Fanuc TP program (LS listing): FM141750.ls

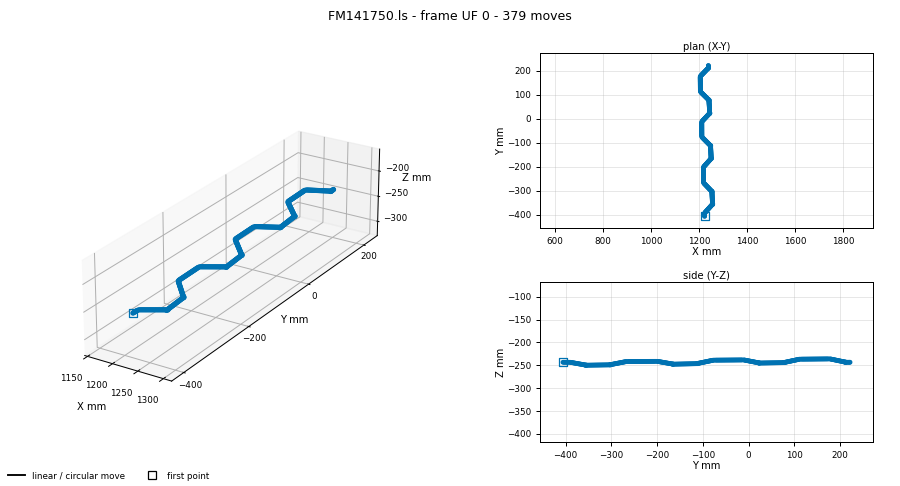
[picture p0: tool path of FM141750.ls in frame UF 0, 379 of 379 moves have a stored position in this frame; points joined in program order, loops and branches not executed]
/PROG  FM141750
/ATTR
OWNER		= MNEDITOR;
COMMENT		= "Auto FANUC move";
PROG_SIZE	= 0;
CREATE		= DATE 26-05-06  TIME 14:17:50;
MODIFIED	= DATE 26-05-06  TIME 14:17:50;
FILE_NAME	= ;
VERSION		= 0;
LINE_COUNT	= 384;
MEMORY_SIZE	= 0;
PROTECT		= READ_WRITE;
TCD:  STACK_SIZE	= 0,
      TASK_PRIORITY	= 50,
      TIME_SLICE	= 0,
      BUSY_LAMP_OFF	= 0,
      ABORT_REQUEST	= 0,
      PAUSE_REQUEST	= 0;
DEFAULT_GROUP	= 1,*,*,*,*;
CONTROL_CODE	= 00000000 00000000;
/MN
   1:  UFRAME_NUM=0 ;
   2:  UTOOL_NUM=1 ;
   3:  R[93]=10 ;
   4:  L P[1] 7mm/sec FINE ;
   5:  L P[2] 7mm/sec CNT50 ;
   6:  L P[3] 7mm/sec CNT50 ;
   7:  L P[4] 7mm/sec CNT50 ;
   8:  L P[5] 7mm/sec CNT50 ;
   9:  L P[6] 7mm/sec CNT50 ;
  10:  L P[7] 7mm/sec CNT50 ;
  11:  L P[8] 7mm/sec CNT50 ;
  12:  L P[9] 7mm/sec CNT50 ;
  13:  L P[10] 7mm/sec CNT50 ;
  14:  L P[11] 7mm/sec CNT50 ;
  15:  L P[12] 7mm/sec CNT50 ;
  16:  L P[13] 7mm/sec CNT50 ;
  17:  L P[14] 7mm/sec CNT50 ;
  18:  L P[15] 7mm/sec CNT50 ;
  19:  L P[16] 7mm/sec CNT50 ;
  20:  L P[17] 7mm/sec CNT50 ;
  21:  L P[18] 7mm/sec CNT50 ;
  22:  L P[19] 7mm/sec CNT50 ;
  23:  L P[20] 7mm/sec CNT50 ;
  24:  L P[21] 7mm/sec CNT50 ;
  25:  L P[22] 7mm/sec CNT50 ;
  26:  L P[23] 7mm/sec CNT50 ;
  27:  L P[24] 7mm/sec CNT50 ;
  28:  L P[25] 7mm/sec CNT50 ;
  29:  L P[26] 7mm/sec CNT50 ;
  30:  L P[27] 7mm/sec CNT50 ;
  31:  L P[28] 7mm/sec CNT50 ;
  32:  L P[29] 7mm/sec CNT50 ;
  33:  L P[30] 7mm/sec CNT50 ;
  34:  L P[31] 7mm/sec CNT50 ;
  35:  L P[32] 7mm/sec CNT50 ;
  36:  L P[33] 7mm/sec CNT50 ;
  37:  L P[34] 7mm/sec CNT50 ;
  38:  L P[35] 7mm/sec CNT50 ;
  39:  L P[36] 7mm/sec CNT50 ;
  40:  L P[37] 7mm/sec CNT50 ;
  41:  L P[38] 7mm/sec CNT50 ;
  42:  L P[39] 7mm/sec CNT50 ;
  43:  L P[40] 7mm/sec CNT50 ;
  44:  L P[41] 7mm/sec CNT50 ;
  45:  L P[42] 7mm/sec CNT50 ;
  46:  L P[43] 7mm/sec CNT50 ;
  47:  L P[44] 7mm/sec CNT50 ;
  48:  L P[45] 7mm/sec CNT50 ;
  49:  L P[46] 7mm/sec CNT50 ;
  50:  L P[47] 7mm/sec CNT50 ;
  51:  L P[48] 7mm/sec CNT50 ;
  52:  L P[49] 7mm/sec CNT50 ;
  53:  L P[50] 7mm/sec CNT50 ;
  54:  L P[51] 7mm/sec CNT50 ;
  55:  L P[52] 7mm/sec CNT50 ;
  56:  L P[53] 7mm/sec CNT50 ;
  57:  L P[54] 7mm/sec CNT50 ;
  58:  L P[55] 7mm/sec CNT50 ;
  59:  L P[56] 7mm/sec CNT50 ;
  60:  L P[57] 7mm/sec CNT50 ;
  61:  L P[58] 7mm/sec CNT50 ;
  62:  L P[59] 7mm/sec CNT50 ;
  63:  L P[60] 7mm/sec CNT50 ;
  64:  L P[61] 7mm/sec CNT50 ;
  65:  L P[62] 7mm/sec CNT50 ;
  66:  L P[63] 7mm/sec CNT50 ;
  67:  L P[64] 7mm/sec CNT50 ;
  68:  L P[65] 7mm/sec CNT50 ;
  69:  L P[66] 7mm/sec CNT50 ;
  70:  L P[67] 7mm/sec CNT50 ;
  71:  L P[68] 7mm/sec CNT50 ;
  72:  L P[69] 7mm/sec CNT50 ;
  73:  L P[70] 7mm/sec CNT50 ;
  74:  L P[71] 7mm/sec CNT50 ;
  75:  L P[72] 7mm/sec CNT50 ;
  76:  L P[73] 7mm/sec CNT50 ;
  77:  L P[74] 7mm/sec CNT50 ;
  78:  L P[75] 7mm/sec CNT50 ;
  79:  L P[76] 7mm/sec CNT50 ;
  80:  L P[77] 7mm/sec CNT50 ;
  81:  L P[78] 7mm/sec CNT50 ;
  82:  L P[79] 7mm/sec CNT50 ;
  83:  L P[80] 7mm/sec CNT50 ;
  84:  L P[81] 7mm/sec CNT50 ;
  85:  L P[82] 7mm/sec CNT50 ;
  86:  L P[83] 7mm/sec CNT50 ;
  87:  L P[84] 7mm/sec CNT50 ;
  88:  L P[85] 7mm/sec CNT50 ;
  89:  L P[86] 7mm/sec CNT50 ;
  90:  L P[87] 7mm/sec CNT50 ;
  91:  L P[88] 7mm/sec CNT50 ;
  92:  L P[89] 7mm/sec CNT50 ;
  93:  L P[90] 7mm/sec CNT50 ;
  94:  L P[91] 7mm/sec CNT50 ;
  95:  L P[92] 7mm/sec CNT50 ;
  96:  L P[93] 7mm/sec CNT50 ;
  97:  L P[94] 7mm/sec CNT50 ;
  98:  L P[95] 7mm/sec CNT50 ;
  99:  L P[96] 7mm/sec CNT50 ;
 100:  L P[97] 7mm/sec CNT50 ;
 101:  L P[98] 7mm/sec CNT50 ;
 102:  L P[99] 7mm/sec CNT50 ;
 103:  L P[100] 7mm/sec CNT50 ;
 104:  L P[101] 7mm/sec CNT50 ;
 105:  L P[102] 7mm/sec CNT50 ;
 106:  L P[103] 7mm/sec CNT50 ;
 107:  L P[104] 7mm/sec CNT50 ;
 108:  L P[105] 7mm/sec CNT50 ;
 109:  L P[106] 7mm/sec CNT50 ;
 110:  L P[107] 7mm/sec CNT50 ;
 111:  L P[108] 7mm/sec CNT50 ;
 112:  L P[109] 7mm/sec CNT50 ;
 113:  L P[110] 7mm/sec CNT50 ;
 114:  L P[111] 7mm/sec CNT50 ;
 115:  L P[112] 7mm/sec CNT50 ;
 116:  L P[113] 7mm/sec CNT50 ;
 117:  L P[114] 7mm/sec CNT50 ;
 118:  L P[115] 7mm/sec CNT50 ;
 119:  L P[116] 7mm/sec CNT50 ;
 120:  L P[117] 7mm/sec CNT50 ;
 121:  L P[118] 7mm/sec CNT50 ;
 122:  L P[119] 7mm/sec CNT50 ;
 123:  L P[120] 7mm/sec CNT50 ;
 124:  L P[121] 7mm/sec CNT50 ;
 125:  L P[122] 7mm/sec CNT50 ;
 126:  L P[123] 7mm/sec CNT50 ;
 127:  L P[124] 7mm/sec CNT50 ;
 128:  L P[125] 7mm/sec CNT50 ;
 129:  L P[126] 7mm/sec CNT50 ;
 130:  L P[127] 7mm/sec CNT50 ;
 131:  L P[128] 7mm/sec CNT50 ;
 132:  L P[129] 7mm/sec CNT50 ;
 133:  L P[130] 7mm/sec CNT50 ;
 134:  L P[131] 7mm/sec CNT50 ;
 135:  L P[132] 7mm/sec CNT50 ;
 136:  L P[133] 7mm/sec CNT50 ;
 137:  L P[134] 7mm/sec CNT50 ;
 138:  L P[135] 7mm/sec CNT50 ;
 139:  L P[136] 7mm/sec CNT50 ;
 140:  L P[137] 7mm/sec CNT50 ;
 141:  L P[138] 7mm/sec CNT50 ;
 142:  L P[139] 7mm/sec CNT50 ;
 143:  L P[140] 7mm/sec CNT50 ;
 144:  L P[141] 7mm/sec CNT50 ;
 145:  L P[142] 7mm/sec CNT50 ;
 146:  L P[143] 7mm/sec CNT50 ;
 147:  L P[144] 7mm/sec CNT50 ;
 148:  L P[145] 7mm/sec CNT50 ;
 149:  L P[146] 7mm/sec CNT50 ;
 150:  L P[147] 7mm/sec CNT50 ;
 151:  L P[148] 7mm/sec CNT50 ;
 152:  L P[149] 7mm/sec CNT50 ;
 153:  L P[150] 7mm/sec CNT50 ;
 154:  L P[151] 7mm/sec CNT50 ;
 155:  L P[152] 7mm/sec CNT50 ;
 156:  L P[153] 7mm/sec CNT50 ;
 157:  L P[154] 7mm/sec CNT50 ;
 158:  L P[155] 7mm/sec CNT50 ;
 159:  L P[156] 7mm/sec CNT50 ;
 160:  L P[157] 7mm/sec CNT50 ;
 161:  L P[158] 7mm/sec CNT50 ;
 162:  L P[159] 7mm/sec CNT50 ;
 163:  L P[160] 7mm/sec CNT50 ;
 164:  L P[161] 7mm/sec CNT50 ;
 165:  L P[162] 7mm/sec CNT50 ;
 166:  L P[163] 7mm/sec CNT50 ;
 167:  L P[164] 7mm/sec CNT50 ;
 168:  L P[165] 7mm/sec CNT50 ;
 169:  L P[166] 7mm/sec CNT50 ;
 170:  L P[167] 7mm/sec CNT50 ;
 171:  L P[168] 7mm/sec CNT50 ;
 172:  L P[169] 7mm/sec CNT50 ;
 173:  L P[170] 7mm/sec CNT50 ;
 174:  L P[171] 7mm/sec CNT50 ;
 175:  L P[172] 7mm/sec CNT50 ;
 176:  L P[173] 7mm/sec CNT50 ;
 177:  L P[174] 7mm/sec CNT50 ;
 178:  L P[175] 7mm/sec CNT50 ;
 179:  L P[176] 7mm/sec CNT50 ;
 180:  L P[177] 7mm/sec CNT50 ;
 181:  L P[178] 7mm/sec CNT50 ;
 182:  L P[179] 7mm/sec CNT50 ;
 183:  L P[180] 7mm/sec CNT50 ;
 184:  L P[181] 7mm/sec CNT50 ;
 185:  L P[182] 7mm/sec CNT50 ;
 186:  L P[183] 7mm/sec CNT50 ;
 187:  L P[184] 7mm/sec CNT50 ;
 188:  L P[185] 7mm/sec CNT50 ;
 189:  L P[186] 7mm/sec CNT50 ;
 190:  L P[187] 7mm/sec CNT50 ;
 191:  L P[188] 7mm/sec CNT50 ;
 192:  L P[189] 7mm/sec CNT50 ;
 193:  L P[190] 7mm/sec CNT50 ;
 194:  L P[191] 7mm/sec CNT50 ;
 195:  L P[192] 7mm/sec CNT50 ;
 196:  L P[193] 7mm/sec CNT50 ;
 197:  L P[194] 7mm/sec CNT50 ;
 198:  L P[195] 7mm/sec CNT50 ;
 199:  L P[196] 7mm/sec CNT50 ;
 200:  L P[197] 7mm/sec CNT50 ;
 201:  L P[198] 7mm/sec CNT50 ;
 202:  L P[199] 7mm/sec CNT50 ;
 203:  L P[200] 7mm/sec CNT50 ;
 204:  L P[201] 7mm/sec CNT50 ;
 205:  L P[202] 7mm/sec CNT50 ;
 206:  L P[203] 7mm/sec CNT50 ;
 207:  L P[204] 7mm/sec CNT50 ;
 208:  L P[205] 7mm/sec CNT50 ;
 209:  L P[206] 7mm/sec CNT50 ;
 210:  L P[207] 7mm/sec CNT50 ;
 211:  L P[208] 7mm/sec CNT50 ;
 212:  L P[209] 7mm/sec CNT50 ;
 213:  L P[210] 7mm/sec CNT50 ;
 214:  L P[211] 7mm/sec CNT50 ;
 215:  L P[212] 7mm/sec CNT50 ;
 216:  L P[213] 7mm/sec CNT50 ;
 217:  L P[214] 7mm/sec CNT50 ;
 218:  L P[215] 7mm/sec CNT50 ;
 219:  L P[216] 7mm/sec CNT50 ;
 220:  L P[217] 7mm/sec CNT50 ;
 221:  L P[218] 7mm/sec CNT50 ;
 222:  L P[219] 7mm/sec CNT50 ;
 223:  L P[220] 7mm/sec CNT50 ;
 224:  L P[221] 7mm/sec CNT50 ;
 225:  L P[222] 7mm/sec CNT50 ;
 226:  L P[223] 7mm/sec CNT50 ;
 227:  L P[224] 7mm/sec CNT50 ;
 228:  L P[225] 7mm/sec CNT50 ;
 229:  L P[226] 7mm/sec CNT50 ;
 230:  L P[227] 7mm/sec CNT50 ;
 231:  L P[228] 7mm/sec CNT50 ;
 232:  L P[229] 7mm/sec CNT50 ;
 233:  L P[230] 7mm/sec CNT50 ;
 234:  L P[231] 7mm/sec CNT50 ;
 235:  L P[232] 7mm/sec CNT50 ;
 236:  L P[233] 7mm/sec CNT50 ;
 237:  L P[234] 7mm/sec CNT50 ;
 238:  L P[235] 7mm/sec CNT50 ;
 239:  L P[236] 7mm/sec CNT50 ;
 240:  L P[237] 7mm/sec CNT50 ;
 241:  L P[238] 7mm/sec CNT50 ;
 242:  L P[239] 7mm/sec CNT50 ;
 243:  L P[240] 7mm/sec CNT50 ;
 244:  L P[241] 7mm/sec CNT50 ;
 245:  L P[242] 7mm/sec CNT50 ;
 246:  L P[243] 7mm/sec CNT50 ;
 247:  L P[244] 7mm/sec CNT50 ;
 248:  L P[245] 7mm/sec CNT50 ;
 249:  L P[246] 7mm/sec CNT50 ;
 250:  L P[247] 7mm/sec CNT50 ;
 251:  L P[248] 7mm/sec CNT50 ;
 252:  L P[249] 7mm/sec CNT50 ;
 253:  L P[250] 7mm/sec CNT50 ;
 254:  L P[251] 7mm/sec CNT50 ;
 255:  L P[252] 7mm/sec CNT50 ;
 256:  L P[253] 7mm/sec CNT50 ;
 257:  L P[254] 7mm/sec CNT50 ;
 258:  L P[255] 7mm/sec CNT50 ;
 259:  L P[256] 7mm/sec CNT50 ;
 260:  L P[257] 7mm/sec CNT50 ;
 261:  L P[258] 7mm/sec CNT50 ;
 262:  L P[259] 7mm/sec CNT50 ;
 263:  L P[260] 7mm/sec CNT50 ;
 264:  L P[261] 7mm/sec CNT50 ;
 265:  L P[262] 7mm/sec CNT50 ;
 266:  L P[263] 7mm/sec CNT50 ;
 267:  L P[264] 7mm/sec CNT50 ;
 268:  L P[265] 7mm/sec CNT50 ;
 269:  L P[266] 7mm/sec CNT50 ;
 270:  L P[267] 7mm/sec CNT50 ;
 271:  L P[268] 7mm/sec CNT50 ;
 272:  L P[269] 7mm/sec CNT50 ;
 273:  L P[270] 7mm/sec CNT50 ;
 274:  L P[271] 7mm/sec CNT50 ;
 275:  L P[272] 7mm/sec CNT50 ;
 276:  L P[273] 7mm/sec CNT50 ;
 277:  L P[274] 7mm/sec CNT50 ;
 278:  L P[275] 7mm/sec CNT50 ;
 279:  L P[276] 7mm/sec CNT50 ;
 280:  L P[277] 7mm/sec CNT50 ;
 281:  L P[278] 7mm/sec CNT50 ;
 282:  L P[279] 7mm/sec CNT50 ;
 283:  L P[280] 7mm/sec CNT50 ;
 284:  L P[281] 7mm/sec CNT50 ;
 285:  L P[282] 7mm/sec CNT50 ;
 286:  L P[283] 7mm/sec CNT50 ;
 287:  L P[284] 7mm/sec CNT50 ;
 288:  L P[285] 7mm/sec CNT50 ;
 289:  L P[286] 7mm/sec CNT50 ;
 290:  L P[287] 7mm/sec CNT50 ;
 291:  L P[288] 7mm/sec CNT50 ;
 292:  L P[289] 7mm/sec CNT50 ;
 293:  L P[290] 7mm/sec CNT50 ;
 294:  L P[291] 7mm/sec CNT50 ;
 295:  L P[292] 7mm/sec CNT50 ;
 296:  L P[293] 7mm/sec CNT50 ;
 297:  L P[294] 7mm/sec CNT50 ;
 298:  L P[295] 7mm/sec CNT50 ;
 299:  L P[296] 7mm/sec CNT50 ;
 300:  L P[297] 7mm/sec CNT50 ;
 301:  L P[298] 7mm/sec CNT50 ;
 302:  L P[299] 7mm/sec CNT50 ;
 303:  L P[300] 7mm/sec CNT50 ;
 304:  L P[301] 7mm/sec CNT50 ;
 305:  L P[302] 7mm/sec CNT50 ;
 306:  L P[303] 7mm/sec CNT50 ;
 307:  L P[304] 7mm/sec CNT50 ;
 308:  L P[305] 7mm/sec CNT50 ;
 309:  L P[306] 7mm/sec CNT50 ;
 310:  L P[307] 7mm/sec CNT50 ;
 311:  L P[308] 7mm/sec CNT50 ;
 312:  L P[309] 7mm/sec CNT50 ;
 313:  L P[310] 7mm/sec CNT50 ;
 314:  L P[311] 7mm/sec CNT50 ;
 315:  L P[312] 7mm/sec CNT50 ;
 316:  L P[313] 7mm/sec CNT50 ;
 317:  L P[314] 7mm/sec CNT50 ;
 318:  L P[315] 7mm/sec CNT50 ;
 319:  L P[316] 7mm/sec CNT50 ;
 320:  L P[317] 7mm/sec CNT50 ;
 321:  L P[318] 7mm/sec CNT50 ;
 322:  L P[319] 7mm/sec CNT50 ;
 323:  L P[320] 7mm/sec CNT50 ;
 324:  L P[321] 7mm/sec CNT50 ;
 325:  L P[322] 7mm/sec CNT50 ;
 326:  L P[323] 7mm/sec CNT50 ;
 327:  L P[324] 7mm/sec CNT50 ;
 328:  L P[325] 7mm/sec CNT50 ;
 329:  L P[326] 7mm/sec CNT50 ;
 330:  L P[327] 7mm/sec CNT50 ;
 331:  L P[328] 7mm/sec CNT50 ;
 332:  L P[329] 7mm/sec CNT50 ;
 333:  L P[330] 7mm/sec CNT50 ;
 334:  L P[331] 7mm/sec CNT50 ;
 335:  L P[332] 7mm/sec CNT50 ;
 336:  L P[333] 7mm/sec CNT50 ;
 337:  L P[334] 7mm/sec CNT50 ;
 338:  L P[335] 7mm/sec CNT50 ;
 339:  L P[336] 7mm/sec CNT50 ;
 340:  L P[337] 7mm/sec CNT50 ;
 341:  L P[338] 7mm/sec CNT50 ;
 342:  L P[339] 7mm/sec CNT50 ;
 343:  L P[340] 7mm/sec CNT50 ;
 344:  L P[341] 7mm/sec CNT50 ;
 345:  L P[342] 7mm/sec CNT50 ;
 346:  L P[343] 7mm/sec CNT50 ;
 347:  L P[344] 7mm/sec CNT50 ;
 348:  L P[345] 7mm/sec CNT50 ;
 349:  L P[346] 7mm/sec CNT50 ;
 350:  L P[347] 7mm/sec CNT50 ;
 351:  L P[348] 7mm/sec CNT50 ;
 352:  L P[349] 7mm/sec CNT50 ;
 353:  L P[350] 7mm/sec CNT50 ;
 354:  L P[351] 7mm/sec CNT50 ;
 355:  L P[352] 7mm/sec CNT50 ;
 356:  L P[353] 7mm/sec CNT50 ;
 357:  L P[354] 7mm/sec CNT50 ;
 358:  L P[355] 7mm/sec CNT50 ;
 359:  L P[356] 7mm/sec CNT50 ;
 360:  L P[357] 7mm/sec CNT50 ;
 361:  L P[358] 7mm/sec CNT50 ;
 362:  L P[359] 7mm/sec CNT50 ;
 363:  L P[360] 7mm/sec CNT50 ;
 364:  L P[361] 7mm/sec CNT50 ;
 365:  L P[362] 7mm/sec CNT50 ;
 366:  L P[363] 7mm/sec CNT50 ;
 367:  L P[364] 7mm/sec CNT50 ;
 368:  L P[365] 7mm/sec CNT50 ;
 369:  L P[366] 7mm/sec CNT50 ;
 370:  L P[367] 7mm/sec CNT50 ;
 371:  L P[368] 7mm/sec CNT50 ;
 372:  L P[369] 7mm/sec CNT50 ;
 373:  L P[370] 7mm/sec CNT50 ;
 374:  L P[371] 7mm/sec CNT50 ;
 375:  L P[372] 7mm/sec CNT50 ;
 376:  L P[373] 7mm/sec CNT50 ;
 377:  L P[374] 7mm/sec CNT50 ;
 378:  L P[375] 7mm/sec CNT50 ;
 379:  L P[376] 7mm/sec CNT50 ;
 380:  L P[377] 7mm/sec CNT50 ;
 381:  L P[378] 7mm/sec CNT50 ;
 382:  L P[379] 7mm/sec FINE ;
 383:  R[93]=1 ;
 384:  END ;
/POS
P[1]{
   GP1:
	UF : 0, UT : 1,		CONFIG : 'N U T, 0, 0, 0',
	X = 1222.210  mm,	Y = -405.958  mm,	Z = -243.379  mm,
	W = 0.000 deg,	P = 30.000 deg,	R = 178.529 deg
};
P[2]{
   GP1:
	UF : 0, UT : 1,		CONFIG : 'N U T, 0, 0, 0',
	X = 1222.261  mm,	Y = -403.959  mm,	Z = -243.380  mm,
	W = 0.000 deg,	P = 30.000 deg,	R = 178.529 deg
};
P[3]{
   GP1:
	UF : 0, UT : 1,		CONFIG : 'N U T, 0, 0, 0',
	X = 1222.312  mm,	Y = -401.960  mm,	Z = -243.381  mm,
	W = 0.000 deg,	P = 30.000 deg,	R = 170.399 deg
};
P[4]{
   GP1:
	UF : 0, UT : 1,		CONFIG : 'N U T, 0, 0, 0',
	X = 1222.364  mm,	Y = -399.960  mm,	Z = -243.383  mm,
	W = 0.000 deg,	P = 30.000 deg,	R = 162.269 deg
};
P[5]{
   GP1:
	UF : 0, UT : 1,		CONFIG : 'N U T, 0, 0, 0',
	X = 1222.415  mm,	Y = -397.961  mm,	Z = -243.384  mm,
	W = 0.000 deg,	P = 30.000 deg,	R = 154.139 deg
};
P[6]{
   GP1:
	UF : 0, UT : 1,		CONFIG : 'N U T, 0, 0, 0',
	X = 1222.466  mm,	Y = -395.962  mm,	Z = -243.385  mm,
	W = 0.000 deg,	P = 30.000 deg,	R = 146.009 deg
};
P[7]{
   GP1:
	UF : 0, UT : 1,		CONFIG : 'N U T, 0, 0, 0',
	X = 1222.518  mm,	Y = -393.962  mm,	Z = -243.387  mm,
	W = 0.000 deg,	P = 30.000 deg,	R = 137.880 deg
};
P[8]{
   GP1:
	UF : 0, UT : 1,		CONFIG : 'N U T, 0, 0, 0',
	X = 1223.380  mm,	Y = -390.882  mm,	Z = -243.387  mm,
	W = 0.000 deg,	P = 30.000 deg,	R = 137.880 deg
};
P[9]{
   GP1:
	UF : 0, UT : 1,		CONFIG : 'N U T, 0, 0, 0',
	X = 1224.872  mm,	Y = -389.157  mm,	Z = -243.595  mm,
	W = 0.000 deg,	P = 30.000 deg,	R = 137.880 deg
};
P[10]{
   GP1:
	UF : 0, UT : 1,		CONFIG : 'N U T, 0, 0, 0',
	X = 1226.202  mm,	Y = -387.686  mm,	Z = -243.857  mm,
	W = 0.000 deg,	P = 30.000 deg,	R = 137.880 deg
};
P[11]{
   GP1:
	UF : 0, UT : 1,		CONFIG : 'N U T, 0, 0, 0',
	X = 1227.531  mm,	Y = -386.216  mm,	Z = -244.119  mm,
	W = 0.000 deg,	P = 30.000 deg,	R = 137.880 deg
};
P[12]{
   GP1:
	UF : 0, UT : 1,		CONFIG : 'N U T, 0, 0, 0',
	X = 1228.861  mm,	Y = -384.745  mm,	Z = -244.381  mm,
	W = 0.000 deg,	P = 30.000 deg,	R = 137.880 deg
};
P[13]{
   GP1:
	UF : 0, UT : 1,		CONFIG : 'N U T, 0, 0, 0',
	X = 1230.191  mm,	Y = -383.274  mm,	Z = -244.643  mm,
	W = 0.000 deg,	P = 30.000 deg,	R = 137.880 deg
};
P[14]{
   GP1:
	UF : 0, UT : 1,		CONFIG : 'N U T, 0, 0, 0',
	X = 1231.521  mm,	Y = -381.804  mm,	Z = -244.905  mm,
	W = 0.000 deg,	P = 30.000 deg,	R = 137.880 deg
};
P[15]{
   GP1:
	UF : 0, UT : 1,		CONFIG : 'N U T, 0, 0, 0',
	X = 1232.851  mm,	Y = -380.333  mm,	Z = -245.167  mm,
	W = 0.000 deg,	P = 30.000 deg,	R = 137.880 deg
};
P[16]{
   GP1:
	UF : 0, UT : 1,		CONFIG : 'N U T, 0, 0, 0',
	X = 1234.181  mm,	Y = -378.862  mm,	Z = -245.429  mm,
	W = 0.000 deg,	P = 30.000 deg,	R = 137.880 deg
};
P[17]{
   GP1:
	UF : 0, UT : 1,		CONFIG : 'N U T, 0, 0, 0',
	X = 1235.510  mm,	Y = -377.392  mm,	Z = -245.692  mm,
	W = 0.000 deg,	P = 30.000 deg,	R = 137.880 deg
};
P[18]{
   GP1:
	UF : 0, UT : 1,		CONFIG : 'N U T, 0, 0, 0',
	X = 1236.840  mm,	Y = -375.921  mm,	Z = -245.954  mm,
	W = 0.000 deg,	P = 30.000 deg,	R = 137.880 deg
};
P[19]{
   GP1:
	UF : 0, UT : 1,		CONFIG : 'N U T, 0, 0, 0',
	X = 1238.170  mm,	Y = -374.450  mm,	Z = -246.216  mm,
	W = 0.000 deg,	P = 30.000 deg,	R = 137.880 deg
};
P[20]{
   GP1:
	UF : 0, UT : 1,		CONFIG : 'N U T, 0, 0, 0',
	X = 1239.500  mm,	Y = -372.979  mm,	Z = -246.478  mm,
	W = 0.000 deg,	P = 30.000 deg,	R = 137.880 deg
};
P[21]{
   GP1:
	UF : 0, UT : 1,		CONFIG : 'N U T, 0, 0, 0',
	X = 1240.830  mm,	Y = -371.509  mm,	Z = -246.740  mm,
	W = 0.000 deg,	P = 30.000 deg,	R = 137.880 deg
};
P[22]{
   GP1:
	UF : 0, UT : 1,		CONFIG : 'N U T, 0, 0, 0',
	X = 1242.159  mm,	Y = -370.038  mm,	Z = -247.002  mm,
	W = 0.000 deg,	P = 30.000 deg,	R = 137.880 deg
};
P[23]{
   GP1:
	UF : 0, UT : 1,		CONFIG : 'N U T, 0, 0, 0',
	X = 1243.489  mm,	Y = -368.567  mm,	Z = -247.264  mm,
	W = 0.000 deg,	P = 30.000 deg,	R = 137.880 deg
};
P[24]{
   GP1:
	UF : 0, UT : 1,		CONFIG : 'N U T, 0, 0, 0',
	X = 1244.819  mm,	Y = -367.097  mm,	Z = -247.526  mm,
	W = 0.000 deg,	P = 30.000 deg,	R = 137.880 deg
};
P[25]{
   GP1:
	UF : 0, UT : 1,		CONFIG : 'N U T, 0, 0, 0',
	X = 1246.149  mm,	Y = -365.626  mm,	Z = -247.789  mm,
	W = 0.000 deg,	P = 30.000 deg,	R = 137.880 deg
};
P[26]{
   GP1:
	UF : 0, UT : 1,		CONFIG : 'N U T, 0, 0, 0',
	X = 1247.479  mm,	Y = -364.155  mm,	Z = -248.051  mm,
	W = 0.000 deg,	P = 30.000 deg,	R = 137.880 deg
};
P[27]{
   GP1:
	UF : 0, UT : 1,		CONFIG : 'N U T, 0, 0, 0',
	X = 1248.808  mm,	Y = -362.685  mm,	Z = -248.313  mm,
	W = 0.000 deg,	P = 30.000 deg,	R = 137.880 deg
};
P[28]{
   GP1:
	UF : 0, UT : 1,		CONFIG : 'N U T, 0, 0, 0',
	X = 1250.138  mm,	Y = -361.214  mm,	Z = -248.575  mm,
	W = 0.000 deg,	P = 30.000 deg,	R = 144.983 deg
};
P[29]{
   GP1:
	UF : 0, UT : 1,		CONFIG : 'N U T, 0, 0, 0',
	X = 1251.468  mm,	Y = -359.743  mm,	Z = -248.837  mm,
	W = 0.000 deg,	P = 30.000 deg,	R = 153.945 deg
};
P[30]{
   GP1:
	UF : 0, UT : 1,		CONFIG : 'N U T, 0, 0, 0',
	X = 1252.798  mm,	Y = -358.273  mm,	Z = -249.099  mm,
	W = 0.000 deg,	P = 30.000 deg,	R = 162.908 deg
};
P[31]{
   GP1:
	UF : 0, UT : 1,		CONFIG : 'N U T, 0, 0, 0',
	X = 1254.128  mm,	Y = -356.802  mm,	Z = -249.361  mm,
	W = 0.000 deg,	P = 30.000 deg,	R = 171.870 deg
};
P[32]{
   GP1:
	UF : 0, UT : 1,		CONFIG : 'N U T, 0, 0, 0',
	X = 1255.458  mm,	Y = -355.331  mm,	Z = -249.623  mm,
	W = 0.000 deg,	P = 30.000 deg,	R = -179.167 deg
};
P[33]{
   GP1:
	UF : 0, UT : 1,		CONFIG : 'N U T, 0, 0, 0',
	X = 1256.228  mm,	Y = -354.527  mm,	Z = -249.845  mm,
	W = 0.000 deg,	P = 30.000 deg,	R = -177.308 deg
};
P[34]{
   GP1:
	UF : 0, UT : 1,		CONFIG : 'N U T, 0, 0, 0',
	X = 1255.284  mm,	Y = -357.368  mm,	Z = -249.841  mm,
	W = 0.000 deg,	P = 30.000 deg,	R = -177.308 deg
};
P[35]{
   GP1:
	UF : 0, UT : 1,		CONFIG : 'N U T, 0, 0, 0',
	X = 1255.190  mm,	Y = -355.371  mm,	Z = -249.809  mm,
	W = 0.000 deg,	P = 30.000 deg,	R = -177.308 deg
};
P[36]{
   GP1:
	UF : 0, UT : 1,		CONFIG : 'N U T, 0, 0, 0',
	X = 1255.096  mm,	Y = -353.373  mm,	Z = -249.778  mm,
	W = 0.000 deg,	P = 30.000 deg,	R = -177.308 deg
};
P[37]{
   GP1:
	UF : 0, UT : 1,		CONFIG : 'N U T, 0, 0, 0',
	X = 1255.002  mm,	Y = -351.376  mm,	Z = -249.746  mm,
	W = 0.000 deg,	P = 30.000 deg,	R = -177.308 deg
};
P[38]{
   GP1:
	UF : 0, UT : 1,		CONFIG : 'N U T, 0, 0, 0',
	X = 1254.908  mm,	Y = -349.378  mm,	Z = -249.715  mm,
	W = 0.000 deg,	P = 30.000 deg,	R = -177.308 deg
};
P[39]{
   GP1:
	UF : 0, UT : 1,		CONFIG : 'N U T, 0, 0, 0',
	X = 1254.814  mm,	Y = -347.381  mm,	Z = -249.684  mm,
	W = 0.000 deg,	P = 30.000 deg,	R = -177.308 deg
};
P[40]{
   GP1:
	UF : 0, UT : 1,		CONFIG : 'N U T, 0, 0, 0',
	X = 1254.720  mm,	Y = -345.383  mm,	Z = -249.652  mm,
	W = 0.000 deg,	P = 30.000 deg,	R = -177.308 deg
};
P[41]{
   GP1:
	UF : 0, UT : 1,		CONFIG : 'N U T, 0, 0, 0',
	X = 1254.626  mm,	Y = -343.386  mm,	Z = -249.621  mm,
	W = 0.000 deg,	P = 30.000 deg,	R = -177.308 deg
};
P[42]{
   GP1:
	UF : 0, UT : 1,		CONFIG : 'N U T, 0, 0, 0',
	X = 1254.532  mm,	Y = -341.388  mm,	Z = -249.589  mm,
	W = 0.000 deg,	P = 30.000 deg,	R = -177.308 deg
};
P[43]{
   GP1:
	UF : 0, UT : 1,		CONFIG : 'N U T, 0, 0, 0',
	X = 1254.438  mm,	Y = -339.390  mm,	Z = -249.558  mm,
	W = 0.000 deg,	P = 30.000 deg,	R = -177.308 deg
};
P[44]{
   GP1:
	UF : 0, UT : 1,		CONFIG : 'N U T, 0, 0, 0',
	X = 1254.344  mm,	Y = -337.393  mm,	Z = -249.526  mm,
	W = 0.000 deg,	P = 30.000 deg,	R = -177.308 deg
};
P[45]{
   GP1:
	UF : 0, UT : 1,		CONFIG : 'N U T, 0, 0, 0',
	X = 1254.250  mm,	Y = -335.395  mm,	Z = -249.495  mm,
	W = 0.000 deg,	P = 30.000 deg,	R = -177.308 deg
};
P[46]{
   GP1:
	UF : 0, UT : 1,		CONFIG : 'N U T, 0, 0, 0',
	X = 1254.156  mm,	Y = -333.398  mm,	Z = -249.464  mm,
	W = 0.000 deg,	P = 30.000 deg,	R = -177.308 deg
};
P[47]{
   GP1:
	UF : 0, UT : 1,		CONFIG : 'N U T, 0, 0, 0',
	X = 1254.063  mm,	Y = -331.400  mm,	Z = -249.432  mm,
	W = 0.000 deg,	P = 30.000 deg,	R = -177.308 deg
};
P[48]{
   GP1:
	UF : 0, UT : 1,		CONFIG : 'N U T, 0, 0, 0',
	X = 1253.969  mm,	Y = -329.403  mm,	Z = -249.401  mm,
	W = 0.000 deg,	P = 30.000 deg,	R = -177.308 deg
};
P[49]{
   GP1:
	UF : 0, UT : 1,		CONFIG : 'N U T, 0, 0, 0',
	X = 1253.875  mm,	Y = -327.405  mm,	Z = -249.369  mm,
	W = 0.000 deg,	P = 30.000 deg,	R = -177.308 deg
};
P[50]{
   GP1:
	UF : 0, UT : 1,		CONFIG : 'N U T, 0, 0, 0',
	X = 1253.781  mm,	Y = -325.408  mm,	Z = -249.338  mm,
	W = 0.000 deg,	P = 30.000 deg,	R = -177.308 deg
};
P[51]{
   GP1:
	UF : 0, UT : 1,		CONFIG : 'N U T, 0, 0, 0',
	X = 1253.687  mm,	Y = -323.410  mm,	Z = -249.307  mm,
	W = 0.000 deg,	P = 30.000 deg,	R = -177.308 deg
};
P[52]{
   GP1:
	UF : 0, UT : 1,		CONFIG : 'N U T, 0, 0, 0',
	X = 1253.593  mm,	Y = -321.413  mm,	Z = -249.275  mm,
	W = 0.000 deg,	P = 30.000 deg,	R = -177.308 deg
};
P[53]{
   GP1:
	UF : 0, UT : 1,		CONFIG : 'N U T, 0, 0, 0',
	X = 1253.499  mm,	Y = -319.415  mm,	Z = -249.244  mm,
	W = 0.000 deg,	P = 30.000 deg,	R = -177.308 deg
};
P[54]{
   GP1:
	UF : 0, UT : 1,		CONFIG : 'N U T, 0, 0, 0',
	X = 1253.405  mm,	Y = -317.417  mm,	Z = -249.212  mm,
	W = 0.000 deg,	P = 30.000 deg,	R = -177.308 deg
};
P[55]{
   GP1:
	UF : 0, UT : 1,		CONFIG : 'N U T, 0, 0, 0',
	X = 1253.311  mm,	Y = -315.420  mm,	Z = -249.181  mm,
	W = 0.000 deg,	P = 30.000 deg,	R = -177.308 deg
};
P[56]{
   GP1:
	UF : 0, UT : 1,		CONFIG : 'N U T, 0, 0, 0',
	X = 1253.217  mm,	Y = -313.422  mm,	Z = -249.149  mm,
	W = 0.000 deg,	P = 30.000 deg,	R = -177.308 deg
};
P[57]{
   GP1:
	UF : 0, UT : 1,		CONFIG : 'N U T, 0, 0, 0',
	X = 1253.123  mm,	Y = -311.425  mm,	Z = -249.118  mm,
	W = 0.000 deg,	P = 30.000 deg,	R = -176.055 deg
};
P[58]{
   GP1:
	UF : 0, UT : 1,		CONFIG : 'N U T, 0, 0, 0',
	X = 1253.029  mm,	Y = -309.427  mm,	Z = -249.087  mm,
	W = 0.000 deg,	P = 30.000 deg,	R = -167.870 deg
};
P[59]{
   GP1:
	UF : 0, UT : 1,		CONFIG : 'N U T, 0, 0, 0',
	X = 1252.935  mm,	Y = -307.430  mm,	Z = -249.055  mm,
	W = 0.000 deg,	P = 30.000 deg,	R = -159.686 deg
};
P[60]{
   GP1:
	UF : 0, UT : 1,		CONFIG : 'N U T, 0, 0, 0',
	X = 1252.841  mm,	Y = -305.432  mm,	Z = -249.024  mm,
	W = 0.000 deg,	P = 30.000 deg,	R = -151.501 deg
};
P[61]{
   GP1:
	UF : 0, UT : 1,		CONFIG : 'N U T, 0, 0, 0',
	X = 1252.748  mm,	Y = -303.435  mm,	Z = -248.992  mm,
	W = 0.000 deg,	P = 30.000 deg,	R = -143.316 deg
};
P[62]{
   GP1:
	UF : 0, UT : 1,		CONFIG : 'N U T, 0, 0, 0',
	X = 1252.654  mm,	Y = -301.437  mm,	Z = -248.961  mm,
	W = 0.000 deg,	P = 30.000 deg,	R = -136.385 deg
};
P[63]{
   GP1:
	UF : 0, UT : 1,		CONFIG : 'N U T, 0, 0, 0',
	X = 1253.415  mm,	Y = -303.360  mm,	Z = -248.952  mm,
	W = 0.000 deg,	P = 30.000 deg,	R = -136.385 deg
};
P[64]{
   GP1:
	UF : 0, UT : 1,		CONFIG : 'N U T, 0, 0, 0',
	X = 1253.009  mm,	Y = -303.064  mm,	Z = -248.748  mm,
	W = 0.000 deg,	P = 30.000 deg,	R = -136.385 deg
};
P[65]{
   GP1:
	UF : 0, UT : 1,		CONFIG : 'N U T, 0, 0, 0',
	X = 1251.643  mm,	Y = -301.630  mm,	Z = -248.467  mm,
	W = 0.000 deg,	P = 30.000 deg,	R = -136.385 deg
};
P[66]{
   GP1:
	UF : 0, UT : 1,		CONFIG : 'N U T, 0, 0, 0',
	X = 1250.277  mm,	Y = -300.197  mm,	Z = -248.186  mm,
	W = 0.000 deg,	P = 30.000 deg,	R = -136.385 deg
};
P[67]{
   GP1:
	UF : 0, UT : 1,		CONFIG : 'N U T, 0, 0, 0',
	X = 1248.911  mm,	Y = -298.763  mm,	Z = -247.905  mm,
	W = 0.000 deg,	P = 30.000 deg,	R = -136.385 deg
};
P[68]{
   GP1:
	UF : 0, UT : 1,		CONFIG : 'N U T, 0, 0, 0',
	X = 1247.545  mm,	Y = -297.330  mm,	Z = -247.624  mm,
	W = 0.000 deg,	P = 30.000 deg,	R = -136.385 deg
};
P[69]{
   GP1:
	UF : 0, UT : 1,		CONFIG : 'N U T, 0, 0, 0',
	X = 1246.179  mm,	Y = -295.896  mm,	Z = -247.343  mm,
	W = 0.000 deg,	P = 30.000 deg,	R = -136.385 deg
};
P[70]{
   GP1:
	UF : 0, UT : 1,		CONFIG : 'N U T, 0, 0, 0',
	X = 1244.813  mm,	Y = -294.462  mm,	Z = -247.062  mm,
	W = 0.000 deg,	P = 30.000 deg,	R = -136.385 deg
};
P[71]{
   GP1:
	UF : 0, UT : 1,		CONFIG : 'N U T, 0, 0, 0',
	X = 1243.447  mm,	Y = -293.029  mm,	Z = -246.781  mm,
	W = 0.000 deg,	P = 30.000 deg,	R = -136.385 deg
};
P[72]{
   GP1:
	UF : 0, UT : 1,		CONFIG : 'N U T, 0, 0, 0',
	X = 1242.081  mm,	Y = -291.595  mm,	Z = -246.501  mm,
	W = 0.000 deg,	P = 30.000 deg,	R = -136.385 deg
};
P[73]{
   GP1:
	UF : 0, UT : 1,		CONFIG : 'N U T, 0, 0, 0',
	X = 1240.715  mm,	Y = -290.161  mm,	Z = -246.220  mm,
	W = 0.000 deg,	P = 30.000 deg,	R = -136.385 deg
};
P[74]{
   GP1:
	UF : 0, UT : 1,		CONFIG : 'N U T, 0, 0, 0',
	X = 1239.349  mm,	Y = -288.728  mm,	Z = -245.939  mm,
	W = 0.000 deg,	P = 30.000 deg,	R = -136.385 deg
};
P[75]{
   GP1:
	UF : 0, UT : 1,		CONFIG : 'N U T, 0, 0, 0',
	X = 1237.983  mm,	Y = -287.294  mm,	Z = -245.658  mm,
	W = 0.000 deg,	P = 30.000 deg,	R = -136.385 deg
};
P[76]{
   GP1:
	UF : 0, UT : 1,		CONFIG : 'N U T, 0, 0, 0',
	X = 1236.617  mm,	Y = -285.861  mm,	Z = -245.377  mm,
	W = 0.000 deg,	P = 30.000 deg,	R = -136.385 deg
};
P[77]{
   GP1:
	UF : 0, UT : 1,		CONFIG : 'N U T, 0, 0, 0',
	X = 1235.252  mm,	Y = -284.427  mm,	Z = -245.096  mm,
	W = 0.000 deg,	P = 30.000 deg,	R = -136.385 deg
};
P[78]{
   GP1:
	UF : 0, UT : 1,		CONFIG : 'N U T, 0, 0, 0',
	X = 1233.886  mm,	Y = -282.993  mm,	Z = -244.815  mm,
	W = 0.000 deg,	P = 30.000 deg,	R = -136.385 deg
};
P[79]{
   GP1:
	UF : 0, UT : 1,		CONFIG : 'N U T, 0, 0, 0',
	X = 1232.520  mm,	Y = -281.560  mm,	Z = -244.534  mm,
	W = 0.000 deg,	P = 30.000 deg,	R = -136.385 deg
};
P[80]{
   GP1:
	UF : 0, UT : 1,		CONFIG : 'N U T, 0, 0, 0',
	X = 1231.154  mm,	Y = -280.126  mm,	Z = -244.253  mm,
	W = 0.000 deg,	P = 30.000 deg,	R = -136.385 deg
};
P[81]{
   GP1:
	UF : 0, UT : 1,		CONFIG : 'N U T, 0, 0, 0',
	X = 1229.788  mm,	Y = -278.692  mm,	Z = -243.972  mm,
	W = 0.000 deg,	P = 30.000 deg,	R = -136.385 deg
};
P[82]{
   GP1:
	UF : 0, UT : 1,		CONFIG : 'N U T, 0, 0, 0',
	X = 1228.422  mm,	Y = -277.259  mm,	Z = -243.691  mm,
	W = 0.000 deg,	P = 30.000 deg,	R = -136.385 deg
};
P[83]{
   GP1:
	UF : 0, UT : 1,		CONFIG : 'N U T, 0, 0, 0',
	X = 1227.056  mm,	Y = -275.825  mm,	Z = -243.410  mm,
	W = 0.000 deg,	P = 30.000 deg,	R = -136.385 deg
};
P[84]{
   GP1:
	UF : 0, UT : 1,		CONFIG : 'N U T, 0, 0, 0',
	X = 1225.690  mm,	Y = -274.392  mm,	Z = -243.129  mm,
	W = 0.000 deg,	P = 30.000 deg,	R = -142.689 deg
};
P[85]{
   GP1:
	UF : 0, UT : 1,		CONFIG : 'N U T, 0, 0, 0',
	X = 1224.324  mm,	Y = -272.958  mm,	Z = -242.848  mm,
	W = 0.000 deg,	P = 30.000 deg,	R = -151.355 deg
};
P[86]{
   GP1:
	UF : 0, UT : 1,		CONFIG : 'N U T, 0, 0, 0',
	X = 1222.958  mm,	Y = -271.524  mm,	Z = -242.567  mm,
	W = 0.000 deg,	P = 30.000 deg,	R = -160.022 deg
};
P[87]{
   GP1:
	UF : 0, UT : 1,		CONFIG : 'N U T, 0, 0, 0',
	X = 1221.592  mm,	Y = -270.091  mm,	Z = -242.287  mm,
	W = 0.000 deg,	P = 30.000 deg,	R = -168.688 deg
};
P[88]{
   GP1:
	UF : 0, UT : 1,		CONFIG : 'N U T, 0, 0, 0',
	X = 1220.226  mm,	Y = -268.657  mm,	Z = -242.006  mm,
	W = 0.000 deg,	P = 30.000 deg,	R = -177.354 deg
};
P[89]{
   GP1:
	UF : 0, UT : 1,		CONFIG : 'N U T, 0, 0, 0',
	X = 1218.705  mm,	Y = -267.011  mm,	Z = -241.770  mm,
	W = 0.000 deg,	P = 30.000 deg,	R = -179.716 deg
};
P[90]{
   GP1:
	UF : 0, UT : 1,		CONFIG : 'N U T, 0, 0, 0',
	X = 1217.699  mm,	Y = -263.708  mm,	Z = -241.768  mm,
	W = 0.000 deg,	P = 30.000 deg,	R = -179.716 deg
};
P[91]{
   GP1:
	UF : 0, UT : 1,		CONFIG : 'N U T, 0, 0, 0',
	X = 1217.689  mm,	Y = -261.708  mm,	Z = -241.753  mm,
	W = 0.000 deg,	P = 30.000 deg,	R = -179.716 deg
};
P[92]{
   GP1:
	UF : 0, UT : 1,		CONFIG : 'N U T, 0, 0, 0',
	X = 1217.679  mm,	Y = -259.708  mm,	Z = -241.738  mm,
	W = 0.000 deg,	P = 30.000 deg,	R = -179.716 deg
};
P[93]{
   GP1:
	UF : 0, UT : 1,		CONFIG : 'N U T, 0, 0, 0',
	X = 1217.669  mm,	Y = -257.708  mm,	Z = -241.724  mm,
	W = 0.000 deg,	P = 30.000 deg,	R = -179.716 deg
};
P[94]{
   GP1:
	UF : 0, UT : 1,		CONFIG : 'N U T, 0, 0, 0',
	X = 1217.660  mm,	Y = -255.708  mm,	Z = -241.709  mm,
	W = 0.000 deg,	P = 30.000 deg,	R = -179.716 deg
};
P[95]{
   GP1:
	UF : 0, UT : 1,		CONFIG : 'N U T, 0, 0, 0',
	X = 1217.650  mm,	Y = -253.708  mm,	Z = -241.694  mm,
	W = 0.000 deg,	P = 30.000 deg,	R = -179.716 deg
};
P[96]{
   GP1:
	UF : 0, UT : 1,		CONFIG : 'N U T, 0, 0, 0',
	X = 1217.640  mm,	Y = -251.708  mm,	Z = -241.680  mm,
	W = 0.000 deg,	P = 30.000 deg,	R = -179.716 deg
};
P[97]{
   GP1:
	UF : 0, UT : 1,		CONFIG : 'N U T, 0, 0, 0',
	X = 1217.630  mm,	Y = -249.708  mm,	Z = -241.665  mm,
	W = 0.000 deg,	P = 30.000 deg,	R = -179.716 deg
};
P[98]{
   GP1:
	UF : 0, UT : 1,		CONFIG : 'N U T, 0, 0, 0',
	X = 1217.620  mm,	Y = -247.708  mm,	Z = -241.650  mm,
	W = 0.000 deg,	P = 30.000 deg,	R = -179.716 deg
};
P[99]{
   GP1:
	UF : 0, UT : 1,		CONFIG : 'N U T, 0, 0, 0',
	X = 1217.610  mm,	Y = -245.708  mm,	Z = -241.636  mm,
	W = 0.000 deg,	P = 30.000 deg,	R = -179.716 deg
};
P[100]{
   GP1:
	UF : 0, UT : 1,		CONFIG : 'N U T, 0, 0, 0',
	X = 1217.600  mm,	Y = -243.709  mm,	Z = -241.621  mm,
	W = 0.000 deg,	P = 30.000 deg,	R = -179.716 deg
};
P[101]{
   GP1:
	UF : 0, UT : 1,		CONFIG : 'N U T, 0, 0, 0',
	X = 1217.590  mm,	Y = -241.709  mm,	Z = -241.606  mm,
	W = 0.000 deg,	P = 30.000 deg,	R = -179.716 deg
};
P[102]{
   GP1:
	UF : 0, UT : 1,		CONFIG : 'N U T, 0, 0, 0',
	X = 1217.580  mm,	Y = -239.709  mm,	Z = -241.592  mm,
	W = 0.000 deg,	P = 30.000 deg,	R = -179.716 deg
};
P[103]{
   GP1:
	UF : 0, UT : 1,		CONFIG : 'N U T, 0, 0, 0',
	X = 1217.570  mm,	Y = -237.709  mm,	Z = -241.577  mm,
	W = 0.000 deg,	P = 30.000 deg,	R = -179.716 deg
};
P[104]{
   GP1:
	UF : 0, UT : 1,		CONFIG : 'N U T, 0, 0, 0',
	X = 1217.560  mm,	Y = -235.709  mm,	Z = -241.562  mm,
	W = 0.000 deg,	P = 30.000 deg,	R = -179.716 deg
};
P[105]{
   GP1:
	UF : 0, UT : 1,		CONFIG : 'N U T, 0, 0, 0',
	X = 1217.550  mm,	Y = -233.709  mm,	Z = -241.548  mm,
	W = 0.000 deg,	P = 30.000 deg,	R = -179.716 deg
};
P[106]{
   GP1:
	UF : 0, UT : 1,		CONFIG : 'N U T, 0, 0, 0',
	X = 1217.540  mm,	Y = -231.709  mm,	Z = -241.533  mm,
	W = 0.000 deg,	P = 30.000 deg,	R = -179.716 deg
};
P[107]{
   GP1:
	UF : 0, UT : 1,		CONFIG : 'N U T, 0, 0, 0',
	X = 1217.530  mm,	Y = -229.709  mm,	Z = -241.518  mm,
	W = 0.000 deg,	P = 30.000 deg,	R = -179.716 deg
};
P[108]{
   GP1:
	UF : 0, UT : 1,		CONFIG : 'N U T, 0, 0, 0',
	X = 1217.521  mm,	Y = -227.709  mm,	Z = -241.504  mm,
	W = 0.000 deg,	P = 30.000 deg,	R = -179.716 deg
};
P[109]{
   GP1:
	UF : 0, UT : 1,		CONFIG : 'N U T, 0, 0, 0',
	X = 1217.511  mm,	Y = -225.709  mm,	Z = -241.489  mm,
	W = 0.000 deg,	P = 30.000 deg,	R = -179.716 deg
};
P[110]{
   GP1:
	UF : 0, UT : 1,		CONFIG : 'N U T, 0, 0, 0',
	X = 1217.501  mm,	Y = -223.709  mm,	Z = -241.474  mm,
	W = 0.000 deg,	P = 30.000 deg,	R = -179.716 deg
};
P[111]{
   GP1:
	UF : 0, UT : 1,		CONFIG : 'N U T, 0, 0, 0',
	X = 1217.491  mm,	Y = -221.709  mm,	Z = -241.460  mm,
	W = 0.000 deg,	P = 30.000 deg,	R = -179.716 deg
};
P[112]{
   GP1:
	UF : 0, UT : 1,		CONFIG : 'N U T, 0, 0, 0',
	X = 1217.481  mm,	Y = -219.709  mm,	Z = -241.445  mm,
	W = 0.000 deg,	P = 30.000 deg,	R = -179.716 deg
};
P[113]{
   GP1:
	UF : 0, UT : 1,		CONFIG : 'N U T, 0, 0, 0',
	X = 1217.471  mm,	Y = -217.710  mm,	Z = -241.430  mm,
	W = 0.000 deg,	P = 30.000 deg,	R = -179.716 deg
};
P[114]{
   GP1:
	UF : 0, UT : 1,		CONFIG : 'N U T, 0, 0, 0',
	X = 1217.461  mm,	Y = -215.710  mm,	Z = -241.416  mm,
	W = 0.000 deg,	P = 30.000 deg,	R = -179.716 deg
};
P[115]{
   GP1:
	UF : 0, UT : 1,		CONFIG : 'N U T, 0, 0, 0',
	X = 1217.451  mm,	Y = -213.710  mm,	Z = -241.401  mm,
	W = 0.000 deg,	P = 30.000 deg,	R = -179.716 deg
};
P[116]{
   GP1:
	UF : 0, UT : 1,		CONFIG : 'N U T, 0, 0, 0',
	X = 1217.441  mm,	Y = -211.710  mm,	Z = -241.386  mm,
	W = 0.000 deg,	P = 30.000 deg,	R = 170.500 deg
};
P[117]{
   GP1:
	UF : 0, UT : 1,		CONFIG : 'N U T, 0, 0, 0',
	X = 1217.431  mm,	Y = -209.710  mm,	Z = -241.372  mm,
	W = 0.000 deg,	P = 30.000 deg,	R = 162.077 deg
};
P[118]{
   GP1:
	UF : 0, UT : 1,		CONFIG : 'N U T, 0, 0, 0',
	X = 1217.421  mm,	Y = -207.710  mm,	Z = -241.357  mm,
	W = 0.000 deg,	P = 30.000 deg,	R = 153.654 deg
};
P[119]{
   GP1:
	UF : 0, UT : 1,		CONFIG : 'N U T, 0, 0, 0',
	X = 1217.411  mm,	Y = -205.710  mm,	Z = -241.342  mm,
	W = 0.000 deg,	P = 30.000 deg,	R = 145.231 deg
};
P[120]{
   GP1:
	UF : 0, UT : 1,		CONFIG : 'N U T, 0, 0, 0',
	X = 1217.401  mm,	Y = -203.710  mm,	Z = -241.328  mm,
	W = 0.000 deg,	P = 30.000 deg,	R = 138.168 deg
};
P[121]{
   GP1:
	UF : 0, UT : 1,		CONFIG : 'N U T, 0, 0, 0',
	X = 1218.033  mm,	Y = -200.635  mm,	Z = -241.323  mm,
	W = 0.000 deg,	P = 30.000 deg,	R = 138.168 deg
};
P[122]{
   GP1:
	UF : 0, UT : 1,		CONFIG : 'N U T, 0, 0, 0',
	X = 1219.590  mm,	Y = -198.713  mm,	Z = -241.502  mm,
	W = 0.000 deg,	P = 30.000 deg,	R = 138.168 deg
};
P[123]{
   GP1:
	UF : 0, UT : 1,		CONFIG : 'N U T, 0, 0, 0',
	X = 1220.913  mm,	Y = -197.235  mm,	Z = -241.760  mm,
	W = 0.000 deg,	P = 30.000 deg,	R = 138.168 deg
};
P[124]{
   GP1:
	UF : 0, UT : 1,		CONFIG : 'N U T, 0, 0, 0',
	X = 1222.236  mm,	Y = -195.757  mm,	Z = -242.018  mm,
	W = 0.000 deg,	P = 30.000 deg,	R = 138.168 deg
};
P[125]{
   GP1:
	UF : 0, UT : 1,		CONFIG : 'N U T, 0, 0, 0',
	X = 1223.558  mm,	Y = -194.280  mm,	Z = -242.277  mm,
	W = 0.000 deg,	P = 30.000 deg,	R = 138.168 deg
};
P[126]{
   GP1:
	UF : 0, UT : 1,		CONFIG : 'N U T, 0, 0, 0',
	X = 1224.881  mm,	Y = -192.802  mm,	Z = -242.535  mm,
	W = 0.000 deg,	P = 30.000 deg,	R = 138.168 deg
};
P[127]{
   GP1:
	UF : 0, UT : 1,		CONFIG : 'N U T, 0, 0, 0',
	X = 1226.204  mm,	Y = -191.324  mm,	Z = -242.793  mm,
	W = 0.000 deg,	P = 30.000 deg,	R = 138.168 deg
};
P[128]{
   GP1:
	UF : 0, UT : 1,		CONFIG : 'N U T, 0, 0, 0',
	X = 1227.527  mm,	Y = -189.846  mm,	Z = -243.051  mm,
	W = 0.000 deg,	P = 30.000 deg,	R = 138.168 deg
};
P[129]{
   GP1:
	UF : 0, UT : 1,		CONFIG : 'N U T, 0, 0, 0',
	X = 1228.849  mm,	Y = -188.369  mm,	Z = -243.309  mm,
	W = 0.000 deg,	P = 30.000 deg,	R = 138.168 deg
};
P[130]{
   GP1:
	UF : 0, UT : 1,		CONFIG : 'N U T, 0, 0, 0',
	X = 1230.172  mm,	Y = -186.891  mm,	Z = -243.567  mm,
	W = 0.000 deg,	P = 30.000 deg,	R = 138.168 deg
};
P[131]{
   GP1:
	UF : 0, UT : 1,		CONFIG : 'N U T, 0, 0, 0',
	X = 1231.495  mm,	Y = -185.413  mm,	Z = -243.825  mm,
	W = 0.000 deg,	P = 30.000 deg,	R = 138.168 deg
};
P[132]{
   GP1:
	UF : 0, UT : 1,		CONFIG : 'N U T, 0, 0, 0',
	X = 1232.818  mm,	Y = -183.935  mm,	Z = -244.084  mm,
	W = 0.000 deg,	P = 30.000 deg,	R = 138.168 deg
};
P[133]{
   GP1:
	UF : 0, UT : 1,		CONFIG : 'N U T, 0, 0, 0',
	X = 1234.140  mm,	Y = -182.458  mm,	Z = -244.342  mm,
	W = 0.000 deg,	P = 30.000 deg,	R = 138.168 deg
};
P[134]{
   GP1:
	UF : 0, UT : 1,		CONFIG : 'N U T, 0, 0, 0',
	X = 1235.463  mm,	Y = -180.980  mm,	Z = -244.600  mm,
	W = 0.000 deg,	P = 30.000 deg,	R = 138.168 deg
};
P[135]{
   GP1:
	UF : 0, UT : 1,		CONFIG : 'N U T, 0, 0, 0',
	X = 1236.786  mm,	Y = -179.502  mm,	Z = -244.858  mm,
	W = 0.000 deg,	P = 30.000 deg,	R = 138.168 deg
};
P[136]{
   GP1:
	UF : 0, UT : 1,		CONFIG : 'N U T, 0, 0, 0',
	X = 1238.109  mm,	Y = -178.024  mm,	Z = -245.116  mm,
	W = 0.000 deg,	P = 30.000 deg,	R = 138.168 deg
};
P[137]{
   GP1:
	UF : 0, UT : 1,		CONFIG : 'N U T, 0, 0, 0',
	X = 1239.431  mm,	Y = -176.547  mm,	Z = -245.374  mm,
	W = 0.000 deg,	P = 30.000 deg,	R = 138.168 deg
};
P[138]{
   GP1:
	UF : 0, UT : 1,		CONFIG : 'N U T, 0, 0, 0',
	X = 1240.754  mm,	Y = -175.069  mm,	Z = -245.632  mm,
	W = 0.000 deg,	P = 30.000 deg,	R = 138.168 deg
};
P[139]{
   GP1:
	UF : 0, UT : 1,		CONFIG : 'N U T, 0, 0, 0',
	X = 1242.077  mm,	Y = -173.591  mm,	Z = -245.890  mm,
	W = 0.000 deg,	P = 30.000 deg,	R = 138.168 deg
};
P[140]{
   GP1:
	UF : 0, UT : 1,		CONFIG : 'N U T, 0, 0, 0',
	X = 1243.400  mm,	Y = -172.113  mm,	Z = -246.149  mm,
	W = 0.000 deg,	P = 30.000 deg,	R = 138.168 deg
};
P[141]{
   GP1:
	UF : 0, UT : 1,		CONFIG : 'N U T, 0, 0, 0',
	X = 1244.722  mm,	Y = -170.636  mm,	Z = -246.407  mm,
	W = 0.000 deg,	P = 30.000 deg,	R = 138.168 deg
};
P[142]{
   GP1:
	UF : 0, UT : 1,		CONFIG : 'N U T, 0, 0, 0',
	X = 1246.045  mm,	Y = -169.158  mm,	Z = -246.665  mm,
	W = 0.000 deg,	P = 30.000 deg,	R = 153.214 deg
};
P[143]{
   GP1:
	UF : 0, UT : 1,		CONFIG : 'N U T, 0, 0, 0',
	X = 1247.368  mm,	Y = -167.680  mm,	Z = -246.923  mm,
	W = 0.000 deg,	P = 30.000 deg,	R = 162.098 deg
};
P[144]{
   GP1:
	UF : 0, UT : 1,		CONFIG : 'N U T, 0, 0, 0',
	X = 1248.691  mm,	Y = -166.202  mm,	Z = -247.181  mm,
	W = 0.000 deg,	P = 30.000 deg,	R = 170.981 deg
};
P[145]{
   GP1:
	UF : 0, UT : 1,		CONFIG : 'N U T, 0, 0, 0',
	X = 1250.013  mm,	Y = -164.725  mm,	Z = -247.439  mm,
	W = 0.000 deg,	P = 30.000 deg,	R = 179.865 deg
};
P[146]{
   GP1:
	UF : 0, UT : 1,		CONFIG : 'N U T, 0, 0, 0',
	X = 1250.181  mm,	Y = -164.776  mm,	Z = -247.612  mm,
	W = 0.000 deg,	P = 30.000 deg,	R = -177.413 deg
};
P[147]{
   GP1:
	UF : 0, UT : 1,		CONFIG : 'N U T, 0, 0, 0',
	X = 1249.597  mm,	Y = -166.635  mm,	Z = -247.597  mm,
	W = 0.000 deg,	P = 30.000 deg,	R = -177.413 deg
};
P[148]{
   GP1:
	UF : 0, UT : 1,		CONFIG : 'N U T, 0, 0, 0',
	X = 1249.507  mm,	Y = -164.637  mm,	Z = -247.553  mm,
	W = 0.000 deg,	P = 30.000 deg,	R = -177.413 deg
};
P[149]{
   GP1:
	UF : 0, UT : 1,		CONFIG : 'N U T, 0, 0, 0',
	X = 1249.417  mm,	Y = -162.640  mm,	Z = -247.509  mm,
	W = 0.000 deg,	P = 30.000 deg,	R = -177.413 deg
};
P[150]{
   GP1:
	UF : 0, UT : 1,		CONFIG : 'N U T, 0, 0, 0',
	X = 1249.327  mm,	Y = -160.642  mm,	Z = -247.465  mm,
	W = 0.000 deg,	P = 30.000 deg,	R = -177.413 deg
};
P[151]{
   GP1:
	UF : 0, UT : 1,		CONFIG : 'N U T, 0, 0, 0',
	X = 1249.236  mm,	Y = -158.645  mm,	Z = -247.421  mm,
	W = 0.000 deg,	P = 30.000 deg,	R = -177.413 deg
};
P[152]{
   GP1:
	UF : 0, UT : 1,		CONFIG : 'N U T, 0, 0, 0',
	X = 1249.146  mm,	Y = -156.647  mm,	Z = -247.377  mm,
	W = 0.000 deg,	P = 30.000 deg,	R = -177.413 deg
};
P[153]{
   GP1:
	UF : 0, UT : 1,		CONFIG : 'N U T, 0, 0, 0',
	X = 1249.056  mm,	Y = -154.650  mm,	Z = -247.333  mm,
	W = 0.000 deg,	P = 30.000 deg,	R = -177.413 deg
};
P[154]{
   GP1:
	UF : 0, UT : 1,		CONFIG : 'N U T, 0, 0, 0',
	X = 1248.966  mm,	Y = -152.652  mm,	Z = -247.289  mm,
	W = 0.000 deg,	P = 30.000 deg,	R = -177.413 deg
};
P[155]{
   GP1:
	UF : 0, UT : 1,		CONFIG : 'N U T, 0, 0, 0',
	X = 1248.875  mm,	Y = -150.655  mm,	Z = -247.245  mm,
	W = 0.000 deg,	P = 30.000 deg,	R = -177.413 deg
};
P[156]{
   GP1:
	UF : 0, UT : 1,		CONFIG : 'N U T, 0, 0, 0',
	X = 1248.785  mm,	Y = -148.657  mm,	Z = -247.202  mm,
	W = 0.000 deg,	P = 30.000 deg,	R = -177.413 deg
};
P[157]{
   GP1:
	UF : 0, UT : 1,		CONFIG : 'N U T, 0, 0, 0',
	X = 1248.695  mm,	Y = -146.660  mm,	Z = -247.158  mm,
	W = 0.000 deg,	P = 30.000 deg,	R = -177.413 deg
};
P[158]{
   GP1:
	UF : 0, UT : 1,		CONFIG : 'N U T, 0, 0, 0',
	X = 1248.604  mm,	Y = -144.663  mm,	Z = -247.114  mm,
	W = 0.000 deg,	P = 30.000 deg,	R = -177.413 deg
};
P[159]{
   GP1:
	UF : 0, UT : 1,		CONFIG : 'N U T, 0, 0, 0',
	X = 1248.514  mm,	Y = -142.665  mm,	Z = -247.070  mm,
	W = 0.000 deg,	P = 30.000 deg,	R = -177.413 deg
};
P[160]{
   GP1:
	UF : 0, UT : 1,		CONFIG : 'N U T, 0, 0, 0',
	X = 1248.424  mm,	Y = -140.668  mm,	Z = -247.026  mm,
	W = 0.000 deg,	P = 30.000 deg,	R = -177.413 deg
};
P[161]{
   GP1:
	UF : 0, UT : 1,		CONFIG : 'N U T, 0, 0, 0',
	X = 1248.334  mm,	Y = -138.670  mm,	Z = -246.982  mm,
	W = 0.000 deg,	P = 30.000 deg,	R = -177.413 deg
};
P[162]{
   GP1:
	UF : 0, UT : 1,		CONFIG : 'N U T, 0, 0, 0',
	X = 1248.243  mm,	Y = -136.673  mm,	Z = -246.938  mm,
	W = 0.000 deg,	P = 30.000 deg,	R = -177.413 deg
};
P[163]{
   GP1:
	UF : 0, UT : 1,		CONFIG : 'N U T, 0, 0, 0',
	X = 1248.153  mm,	Y = -134.675  mm,	Z = -246.894  mm,
	W = 0.000 deg,	P = 30.000 deg,	R = -177.413 deg
};
P[164]{
   GP1:
	UF : 0, UT : 1,		CONFIG : 'N U T, 0, 0, 0',
	X = 1248.063  mm,	Y = -132.678  mm,	Z = -246.850  mm,
	W = 0.000 deg,	P = 30.000 deg,	R = -177.413 deg
};
P[165]{
   GP1:
	UF : 0, UT : 1,		CONFIG : 'N U T, 0, 0, 0',
	X = 1247.973  mm,	Y = -130.680  mm,	Z = -246.806  mm,
	W = 0.000 deg,	P = 30.000 deg,	R = -177.413 deg
};
P[166]{
   GP1:
	UF : 0, UT : 1,		CONFIG : 'N U T, 0, 0, 0',
	X = 1247.882  mm,	Y = -128.683  mm,	Z = -246.762  mm,
	W = 0.000 deg,	P = 30.000 deg,	R = -177.413 deg
};
P[167]{
   GP1:
	UF : 0, UT : 1,		CONFIG : 'N U T, 0, 0, 0',
	X = 1247.792  mm,	Y = -126.685  mm,	Z = -246.718  mm,
	W = 0.000 deg,	P = 30.000 deg,	R = -177.413 deg
};
P[168]{
   GP1:
	UF : 0, UT : 1,		CONFIG : 'N U T, 0, 0, 0',
	X = 1247.702  mm,	Y = -124.688  mm,	Z = -246.674  mm,
	W = 0.000 deg,	P = 30.000 deg,	R = -177.413 deg
};
P[169]{
   GP1:
	UF : 0, UT : 1,		CONFIG : 'N U T, 0, 0, 0',
	X = 1247.612  mm,	Y = -122.690  mm,	Z = -246.630  mm,
	W = 0.000 deg,	P = 30.000 deg,	R = -177.413 deg
};
P[170]{
   GP1:
	UF : 0, UT : 1,		CONFIG : 'N U T, 0, 0, 0',
	X = 1247.521  mm,	Y = -120.693  mm,	Z = -246.586  mm,
	W = 0.000 deg,	P = 30.000 deg,	R = -177.413 deg
};
P[171]{
   GP1:
	UF : 0, UT : 1,		CONFIG : 'N U T, 0, 0, 0',
	X = 1247.431  mm,	Y = -118.695  mm,	Z = -246.542  mm,
	W = 0.000 deg,	P = 30.000 deg,	R = -166.168 deg
};
P[172]{
   GP1:
	UF : 0, UT : 1,		CONFIG : 'N U T, 0, 0, 0',
	X = 1247.341  mm,	Y = -116.698  mm,	Z = -246.498  mm,
	W = 0.000 deg,	P = 30.000 deg,	R = -157.727 deg
};
P[173]{
   GP1:
	UF : 0, UT : 1,		CONFIG : 'N U T, 0, 0, 0',
	X = 1247.251  mm,	Y = -114.700  mm,	Z = -246.454  mm,
	W = 0.000 deg,	P = 30.000 deg,	R = -149.286 deg
};
P[174]{
   GP1:
	UF : 0, UT : 1,		CONFIG : 'N U T, 0, 0, 0',
	X = 1247.160  mm,	Y = -112.703  mm,	Z = -246.410  mm,
	W = 0.000 deg,	P = 30.000 deg,	R = -140.845 deg
};
P[175]{
   GP1:
	UF : 0, UT : 1,		CONFIG : 'N U T, 0, 0, 0',
	X = 1247.070  mm,	Y = -110.705  mm,	Z = -246.366  mm,
	W = 0.000 deg,	P = 30.000 deg,	R = -135.207 deg
};
P[176]{
   GP1:
	UF : 0, UT : 1,		CONFIG : 'N U T, 0, 0, 0',
	X = 1247.859  mm,	Y = -112.664  mm,	Z = -246.354  mm,
	W = 0.000 deg,	P = 30.000 deg,	R = -135.207 deg
};
P[177]{
   GP1:
	UF : 0, UT : 1,		CONFIG : 'N U T, 0, 0, 0',
	X = 1247.487  mm,	Y = -112.432  mm,	Z = -246.144  mm,
	W = 0.000 deg,	P = 30.000 deg,	R = -135.207 deg
};
P[178]{
   GP1:
	UF : 0, UT : 1,		CONFIG : 'N U T, 0, 0, 0',
	X = 1246.093  mm,	Y = -111.028  mm,	Z = -245.853  mm,
	W = 0.000 deg,	P = 30.000 deg,	R = -135.207 deg
};
P[179]{
   GP1:
	UF : 0, UT : 1,		CONFIG : 'N U T, 0, 0, 0',
	X = 1244.699  mm,	Y = -109.624  mm,	Z = -245.562  mm,
	W = 0.000 deg,	P = 30.000 deg,	R = -135.207 deg
};
P[180]{
   GP1:
	UF : 0, UT : 1,		CONFIG : 'N U T, 0, 0, 0',
	X = 1243.305  mm,	Y = -108.220  mm,	Z = -245.271  mm,
	W = 0.000 deg,	P = 30.000 deg,	R = -135.207 deg
};
P[181]{
   GP1:
	UF : 0, UT : 1,		CONFIG : 'N U T, 0, 0, 0',
	X = 1241.910  mm,	Y = -106.816  mm,	Z = -244.980  mm,
	W = 0.000 deg,	P = 30.000 deg,	R = -135.207 deg
};
P[182]{
   GP1:
	UF : 0, UT : 1,		CONFIG : 'N U T, 0, 0, 0',
	X = 1240.516  mm,	Y = -105.411  mm,	Z = -244.689  mm,
	W = 0.000 deg,	P = 30.000 deg,	R = -135.207 deg
};
P[183]{
   GP1:
	UF : 0, UT : 1,		CONFIG : 'N U T, 0, 0, 0',
	X = 1239.122  mm,	Y = -104.007  mm,	Z = -244.398  mm,
	W = 0.000 deg,	P = 30.000 deg,	R = -135.207 deg
};
P[184]{
   GP1:
	UF : 0, UT : 1,		CONFIG : 'N U T, 0, 0, 0',
	X = 1237.728  mm,	Y = -102.603  mm,	Z = -244.107  mm,
	W = 0.000 deg,	P = 30.000 deg,	R = -135.207 deg
};
P[185]{
   GP1:
	UF : 0, UT : 1,		CONFIG : 'N U T, 0, 0, 0',
	X = 1236.334  mm,	Y = -101.199  mm,	Z = -243.816  mm,
	W = 0.000 deg,	P = 30.000 deg,	R = -135.207 deg
};
P[186]{
   GP1:
	UF : 0, UT : 1,		CONFIG : 'N U T, 0, 0, 0',
	X = 1234.940  mm,	Y = -99.795  mm,	Z = -243.525  mm,
	W = 0.000 deg,	P = 30.000 deg,	R = -135.207 deg
};
P[187]{
   GP1:
	UF : 0, UT : 1,		CONFIG : 'N U T, 0, 0, 0',
	X = 1233.546  mm,	Y = -98.390  mm,	Z = -243.234  mm,
	W = 0.000 deg,	P = 30.000 deg,	R = -135.207 deg
};
P[188]{
   GP1:
	UF : 0, UT : 1,		CONFIG : 'N U T, 0, 0, 0',
	X = 1232.152  mm,	Y = -96.986  mm,	Z = -242.943  mm,
	W = 0.000 deg,	P = 30.000 deg,	R = -135.207 deg
};
P[189]{
   GP1:
	UF : 0, UT : 1,		CONFIG : 'N U T, 0, 0, 0',
	X = 1230.758  mm,	Y = -95.582  mm,	Z = -242.652  mm,
	W = 0.000 deg,	P = 30.000 deg,	R = -135.207 deg
};
P[190]{
   GP1:
	UF : 0, UT : 1,		CONFIG : 'N U T, 0, 0, 0',
	X = 1229.364  mm,	Y = -94.178  mm,	Z = -242.361  mm,
	W = 0.000 deg,	P = 30.000 deg,	R = -135.207 deg
};
P[191]{
   GP1:
	UF : 0, UT : 1,		CONFIG : 'N U T, 0, 0, 0',
	X = 1227.970  mm,	Y = -92.773  mm,	Z = -242.070  mm,
	W = 0.000 deg,	P = 30.000 deg,	R = -135.207 deg
};
P[192]{
   GP1:
	UF : 0, UT : 1,		CONFIG : 'N U T, 0, 0, 0',
	X = 1226.575  mm,	Y = -91.369  mm,	Z = -241.779  mm,
	W = 0.000 deg,	P = 30.000 deg,	R = -135.207 deg
};
P[193]{
   GP1:
	UF : 0, UT : 1,		CONFIG : 'N U T, 0, 0, 0',
	X = 1225.181  mm,	Y = -89.965  mm,	Z = -241.488  mm,
	W = 0.000 deg,	P = 30.000 deg,	R = -135.207 deg
};
P[194]{
   GP1:
	UF : 0, UT : 1,		CONFIG : 'N U T, 0, 0, 0',
	X = 1223.787  mm,	Y = -88.561  mm,	Z = -241.197  mm,
	W = 0.000 deg,	P = 30.000 deg,	R = -135.207 deg
};
P[195]{
   GP1:
	UF : 0, UT : 1,		CONFIG : 'N U T, 0, 0, 0',
	X = 1222.393  mm,	Y = -87.157  mm,	Z = -240.906  mm,
	W = 0.000 deg,	P = 30.000 deg,	R = -135.207 deg
};
P[196]{
   GP1:
	UF : 0, UT : 1,		CONFIG : 'N U T, 0, 0, 0',
	X = 1220.999  mm,	Y = -85.752  mm,	Z = -240.615  mm,
	W = 0.000 deg,	P = 30.000 deg,	R = -135.207 deg
};
P[197]{
   GP1:
	UF : 0, UT : 1,		CONFIG : 'N U T, 0, 0, 0',
	X = 1219.605  mm,	Y = -84.348  mm,	Z = -240.324  mm,
	W = 0.000 deg,	P = 30.000 deg,	R = -135.207 deg
};
P[198]{
   GP1:
	UF : 0, UT : 1,		CONFIG : 'N U T, 0, 0, 0',
	X = 1218.211  mm,	Y = -82.944  mm,	Z = -240.033  mm,
	W = 0.000 deg,	P = 30.000 deg,	R = -135.207 deg
};
P[199]{
   GP1:
	UF : 0, UT : 1,		CONFIG : 'N U T, 0, 0, 0',
	X = 1216.817  mm,	Y = -81.540  mm,	Z = -239.742  mm,
	W = 0.000 deg,	P = 30.000 deg,	R = -150.556 deg
};
P[200]{
   GP1:
	UF : 0, UT : 1,		CONFIG : 'N U T, 0, 0, 0',
	X = 1215.423  mm,	Y = -80.135  mm,	Z = -239.451  mm,
	W = 0.000 deg,	P = 30.000 deg,	R = -159.476 deg
};
P[201]{
   GP1:
	UF : 0, UT : 1,		CONFIG : 'N U T, 0, 0, 0',
	X = 1214.029  mm,	Y = -78.731  mm,	Z = -239.160  mm,
	W = 0.000 deg,	P = 30.000 deg,	R = -168.397 deg
};
P[202]{
   GP1:
	UF : 0, UT : 1,		CONFIG : 'N U T, 0, 0, 0',
	X = 1212.635  mm,	Y = -77.327  mm,	Z = -238.869  mm,
	W = 0.000 deg,	P = 30.000 deg,	R = -177.317 deg
};
P[203]{
   GP1:
	UF : 0, UT : 1,		CONFIG : 'N U T, 0, 0, 0',
	X = 1210.859  mm,	Y = -74.803  mm,	Z = -238.747  mm,
	W = 0.000 deg,	P = 30.000 deg,	R = -179.809 deg
};
P[204]{
   GP1:
	UF : 0, UT : 1,		CONFIG : 'N U T, 0, 0, 0',
	X = 1210.598  mm,	Y = -72.070  mm,	Z = -238.738  mm,
	W = 0.000 deg,	P = 30.000 deg,	R = -179.809 deg
};
P[205]{
   GP1:
	UF : 0, UT : 1,		CONFIG : 'N U T, 0, 0, 0',
	X = 1210.591  mm,	Y = -70.070  mm,	Z = -238.722  mm,
	W = 0.000 deg,	P = 30.000 deg,	R = -179.809 deg
};
P[206]{
   GP1:
	UF : 0, UT : 1,		CONFIG : 'N U T, 0, 0, 0',
	X = 1210.584  mm,	Y = -68.070  mm,	Z = -238.705  mm,
	W = 0.000 deg,	P = 30.000 deg,	R = -179.809 deg
};
P[207]{
   GP1:
	UF : 0, UT : 1,		CONFIG : 'N U T, 0, 0, 0',
	X = 1210.578  mm,	Y = -66.070  mm,	Z = -238.689  mm,
	W = 0.000 deg,	P = 30.000 deg,	R = -179.809 deg
};
P[208]{
   GP1:
	UF : 0, UT : 1,		CONFIG : 'N U T, 0, 0, 0',
	X = 1210.571  mm,	Y = -64.070  mm,	Z = -238.673  mm,
	W = 0.000 deg,	P = 30.000 deg,	R = -179.809 deg
};
P[209]{
   GP1:
	UF : 0, UT : 1,		CONFIG : 'N U T, 0, 0, 0',
	X = 1210.564  mm,	Y = -62.070  mm,	Z = -238.656  mm,
	W = 0.000 deg,	P = 30.000 deg,	R = -179.809 deg
};
P[210]{
   GP1:
	UF : 0, UT : 1,		CONFIG : 'N U T, 0, 0, 0',
	X = 1210.558  mm,	Y = -60.070  mm,	Z = -238.640  mm,
	W = 0.000 deg,	P = 30.000 deg,	R = -179.809 deg
};
P[211]{
   GP1:
	UF : 0, UT : 1,		CONFIG : 'N U T, 0, 0, 0',
	X = 1210.551  mm,	Y = -58.070  mm,	Z = -238.624  mm,
	W = 0.000 deg,	P = 30.000 deg,	R = -179.809 deg
};
P[212]{
   GP1:
	UF : 0, UT : 1,		CONFIG : 'N U T, 0, 0, 0',
	X = 1210.544  mm,	Y = -56.070  mm,	Z = -238.608  mm,
	W = 0.000 deg,	P = 30.000 deg,	R = -179.809 deg
};
P[213]{
   GP1:
	UF : 0, UT : 1,		CONFIG : 'N U T, 0, 0, 0',
	X = 1210.538  mm,	Y = -54.070  mm,	Z = -238.591  mm,
	W = 0.000 deg,	P = 30.000 deg,	R = -179.809 deg
};
P[214]{
   GP1:
	UF : 0, UT : 1,		CONFIG : 'N U T, 0, 0, 0',
	X = 1210.531  mm,	Y = -52.070  mm,	Z = -238.575  mm,
	W = 0.000 deg,	P = 30.000 deg,	R = -179.809 deg
};
P[215]{
   GP1:
	UF : 0, UT : 1,		CONFIG : 'N U T, 0, 0, 0',
	X = 1210.524  mm,	Y = -50.070  mm,	Z = -238.559  mm,
	W = 0.000 deg,	P = 30.000 deg,	R = -179.809 deg
};
P[216]{
   GP1:
	UF : 0, UT : 1,		CONFIG : 'N U T, 0, 0, 0',
	X = 1210.518  mm,	Y = -48.070  mm,	Z = -238.543  mm,
	W = 0.000 deg,	P = 30.000 deg,	R = -179.809 deg
};
P[217]{
   GP1:
	UF : 0, UT : 1,		CONFIG : 'N U T, 0, 0, 0',
	X = 1210.511  mm,	Y = -46.071  mm,	Z = -238.526  mm,
	W = 0.000 deg,	P = 30.000 deg,	R = -179.809 deg
};
P[218]{
   GP1:
	UF : 0, UT : 1,		CONFIG : 'N U T, 0, 0, 0',
	X = 1210.504  mm,	Y = -44.071  mm,	Z = -238.510  mm,
	W = 0.000 deg,	P = 30.000 deg,	R = -179.809 deg
};
P[219]{
   GP1:
	UF : 0, UT : 1,		CONFIG : 'N U T, 0, 0, 0',
	X = 1210.498  mm,	Y = -42.071  mm,	Z = -238.494  mm,
	W = 0.000 deg,	P = 30.000 deg,	R = -179.809 deg
};
P[220]{
   GP1:
	UF : 0, UT : 1,		CONFIG : 'N U T, 0, 0, 0',
	X = 1210.491  mm,	Y = -40.071  mm,	Z = -238.478  mm,
	W = 0.000 deg,	P = 30.000 deg,	R = -179.809 deg
};
P[221]{
   GP1:
	UF : 0, UT : 1,		CONFIG : 'N U T, 0, 0, 0',
	X = 1210.484  mm,	Y = -38.071  mm,	Z = -238.461  mm,
	W = 0.000 deg,	P = 30.000 deg,	R = -179.809 deg
};
P[222]{
   GP1:
	UF : 0, UT : 1,		CONFIG : 'N U T, 0, 0, 0',
	X = 1210.477  mm,	Y = -36.071  mm,	Z = -238.445  mm,
	W = 0.000 deg,	P = 30.000 deg,	R = -179.809 deg
};
P[223]{
   GP1:
	UF : 0, UT : 1,		CONFIG : 'N U T, 0, 0, 0',
	X = 1210.471  mm,	Y = -34.071  mm,	Z = -238.429  mm,
	W = 0.000 deg,	P = 30.000 deg,	R = -179.809 deg
};
P[224]{
   GP1:
	UF : 0, UT : 1,		CONFIG : 'N U T, 0, 0, 0',
	X = 1210.464  mm,	Y = -32.071  mm,	Z = -238.412  mm,
	W = 0.000 deg,	P = 30.000 deg,	R = -179.809 deg
};
P[225]{
   GP1:
	UF : 0, UT : 1,		CONFIG : 'N U T, 0, 0, 0',
	X = 1210.457  mm,	Y = -30.071  mm,	Z = -238.396  mm,
	W = 0.000 deg,	P = 30.000 deg,	R = -179.809 deg
};
P[226]{
   GP1:
	UF : 0, UT : 1,		CONFIG : 'N U T, 0, 0, 0',
	X = 1210.451  mm,	Y = -28.071  mm,	Z = -238.380  mm,
	W = 0.000 deg,	P = 30.000 deg,	R = -179.809 deg
};
P[227]{
   GP1:
	UF : 0, UT : 1,		CONFIG : 'N U T, 0, 0, 0',
	X = 1210.444  mm,	Y = -26.071  mm,	Z = -238.364  mm,
	W = 0.000 deg,	P = 30.000 deg,	R = -179.809 deg
};
P[228]{
   GP1:
	UF : 0, UT : 1,		CONFIG : 'N U T, 0, 0, 0',
	X = 1210.437  mm,	Y = -24.071  mm,	Z = -238.347  mm,
	W = 0.000 deg,	P = 30.000 deg,	R = -179.809 deg
};
P[229]{
   GP1:
	UF : 0, UT : 1,		CONFIG : 'N U T, 0, 0, 0',
	X = 1210.431  mm,	Y = -22.071  mm,	Z = -238.331  mm,
	W = 0.000 deg,	P = 30.000 deg,	R = 166.443 deg
};
P[230]{
   GP1:
	UF : 0, UT : 1,		CONFIG : 'N U T, 0, 0, 0',
	X = 1210.424  mm,	Y = -20.072  mm,	Z = -238.315  mm,
	W = 0.000 deg,	P = 30.000 deg,	R = 157.758 deg
};
P[231]{
   GP1:
	UF : 0, UT : 1,		CONFIG : 'N U T, 0, 0, 0',
	X = 1210.417  mm,	Y = -18.072  mm,	Z = -238.299  mm,
	W = 0.000 deg,	P = 30.000 deg,	R = 149.073 deg
};
P[232]{
   GP1:
	UF : 0, UT : 1,		CONFIG : 'N U T, 0, 0, 0',
	X = 1210.411  mm,	Y = -16.072  mm,	Z = -238.282  mm,
	W = 0.000 deg,	P = 30.000 deg,	R = 140.388 deg
};
P[233]{
   GP1:
	UF : 0, UT : 1,		CONFIG : 'N U T, 0, 0, 0',
	X = 1210.404  mm,	Y = -14.072  mm,	Z = -238.266  mm,
	W = 0.000 deg,	P = 30.000 deg,	R = 136.766 deg
};
P[234]{
   GP1:
	UF : 0, UT : 1,		CONFIG : 'N U T, 0, 0, 0',
	X = 1211.547  mm,	Y = -10.691  mm,	Z = -238.265  mm,
	W = 0.000 deg,	P = 30.000 deg,	R = 136.766 deg
};
P[235]{
   GP1:
	UF : 0, UT : 1,		CONFIG : 'N U T, 0, 0, 0',
	X = 1212.994  mm,	Y = -9.137  mm,	Z = -238.519  mm,
	W = 0.000 deg,	P = 30.000 deg,	R = 136.766 deg
};
P[236]{
   GP1:
	UF : 0, UT : 1,		CONFIG : 'N U T, 0, 0, 0',
	X = 1214.350  mm,	Y = -7.694  mm,	Z = -238.800  mm,
	W = 0.000 deg,	P = 30.000 deg,	R = 136.766 deg
};
P[237]{
   GP1:
	UF : 0, UT : 1,		CONFIG : 'N U T, 0, 0, 0',
	X = 1215.706  mm,	Y = -6.251  mm,	Z = -239.080  mm,
	W = 0.000 deg,	P = 30.000 deg,	R = 136.766 deg
};
P[238]{
   GP1:
	UF : 0, UT : 1,		CONFIG : 'N U T, 0, 0, 0',
	X = 1217.063  mm,	Y = -4.809  mm,	Z = -239.361  mm,
	W = 0.000 deg,	P = 30.000 deg,	R = 136.766 deg
};
P[239]{
   GP1:
	UF : 0, UT : 1,		CONFIG : 'N U T, 0, 0, 0',
	X = 1218.419  mm,	Y = -3.366  mm,	Z = -239.641  mm,
	W = 0.000 deg,	P = 30.000 deg,	R = 136.766 deg
};
P[240]{
   GP1:
	UF : 0, UT : 1,		CONFIG : 'N U T, 0, 0, 0',
	X = 1219.776  mm,	Y = -1.923  mm,	Z = -239.922  mm,
	W = 0.000 deg,	P = 30.000 deg,	R = 136.766 deg
};
P[241]{
   GP1:
	UF : 0, UT : 1,		CONFIG : 'N U T, 0, 0, 0',
	X = 1221.132  mm,	Y = -0.480  mm,	Z = -240.202  mm,
	W = 0.000 deg,	P = 30.000 deg,	R = 136.766 deg
};
P[242]{
   GP1:
	UF : 0, UT : 1,		CONFIG : 'N U T, 0, 0, 0',
	X = 1222.488  mm,	Y = 0.962  mm,	Z = -240.482  mm,
	W = 0.000 deg,	P = 30.000 deg,	R = 136.766 deg
};
P[243]{
   GP1:
	UF : 0, UT : 1,		CONFIG : 'N U T, 0, 0, 0',
	X = 1223.845  mm,	Y = 2.405  mm,	Z = -240.763  mm,
	W = 0.000 deg,	P = 30.000 deg,	R = 136.766 deg
};
P[244]{
   GP1:
	UF : 0, UT : 1,		CONFIG : 'N U T, 0, 0, 0',
	X = 1225.201  mm,	Y = 3.848  mm,	Z = -241.043  mm,
	W = 0.000 deg,	P = 30.000 deg,	R = 136.766 deg
};
P[245]{
   GP1:
	UF : 0, UT : 1,		CONFIG : 'N U T, 0, 0, 0',
	X = 1226.558  mm,	Y = 5.291  mm,	Z = -241.324  mm,
	W = 0.000 deg,	P = 30.000 deg,	R = 136.766 deg
};
P[246]{
   GP1:
	UF : 0, UT : 1,		CONFIG : 'N U T, 0, 0, 0',
	X = 1227.914  mm,	Y = 6.733  mm,	Z = -241.604  mm,
	W = 0.000 deg,	P = 30.000 deg,	R = 136.766 deg
};
P[247]{
   GP1:
	UF : 0, UT : 1,		CONFIG : 'N U T, 0, 0, 0',
	X = 1229.271  mm,	Y = 8.176  mm,	Z = -241.884  mm,
	W = 0.000 deg,	P = 30.000 deg,	R = 136.766 deg
};
P[248]{
   GP1:
	UF : 0, UT : 1,		CONFIG : 'N U T, 0, 0, 0',
	X = 1230.627  mm,	Y = 9.619  mm,	Z = -242.165  mm,
	W = 0.000 deg,	P = 30.000 deg,	R = 136.766 deg
};
P[249]{
   GP1:
	UF : 0, UT : 1,		CONFIG : 'N U T, 0, 0, 0',
	X = 1231.983  mm,	Y = 11.062  mm,	Z = -242.445  mm,
	W = 0.000 deg,	P = 30.000 deg,	R = 136.766 deg
};
P[250]{
   GP1:
	UF : 0, UT : 1,		CONFIG : 'N U T, 0, 0, 0',
	X = 1233.340  mm,	Y = 12.504  mm,	Z = -242.726  mm,
	W = 0.000 deg,	P = 30.000 deg,	R = 136.766 deg
};
P[251]{
   GP1:
	UF : 0, UT : 1,		CONFIG : 'N U T, 0, 0, 0',
	X = 1234.696  mm,	Y = 13.947  mm,	Z = -243.006  mm,
	W = 0.000 deg,	P = 30.000 deg,	R = 136.766 deg
};
P[252]{
   GP1:
	UF : 0, UT : 1,		CONFIG : 'N U T, 0, 0, 0',
	X = 1236.053  mm,	Y = 15.390  mm,	Z = -243.287  mm,
	W = 0.000 deg,	P = 30.000 deg,	R = 136.766 deg
};
P[253]{
   GP1:
	UF : 0, UT : 1,		CONFIG : 'N U T, 0, 0, 0',
	X = 1237.409  mm,	Y = 16.832  mm,	Z = -243.567  mm,
	W = 0.000 deg,	P = 30.000 deg,	R = 136.766 deg
};
P[254]{
   GP1:
	UF : 0, UT : 1,		CONFIG : 'N U T, 0, 0, 0',
	X = 1238.766  mm,	Y = 18.275  mm,	Z = -243.847  mm,
	W = 0.000 deg,	P = 30.000 deg,	R = 136.766 deg
};
P[255]{
   GP1:
	UF : 0, UT : 1,		CONFIG : 'N U T, 0, 0, 0',
	X = 1240.122  mm,	Y = 19.718  mm,	Z = -244.128  mm,
	W = 0.000 deg,	P = 30.000 deg,	R = 154.477 deg
};
P[256]{
   GP1:
	UF : 0, UT : 1,		CONFIG : 'N U T, 0, 0, 0',
	X = 1241.478  mm,	Y = 21.161  mm,	Z = -244.408  mm,
	W = 0.000 deg,	P = 30.000 deg,	R = 163.754 deg
};
P[257]{
   GP1:
	UF : 0, UT : 1,		CONFIG : 'N U T, 0, 0, 0',
	X = 1242.835  mm,	Y = 22.603  mm,	Z = -244.689  mm,
	W = 0.000 deg,	P = 30.000 deg,	R = 173.032 deg
};
P[258]{
   GP1:
	UF : 0, UT : 1,		CONFIG : 'N U T, 0, 0, 0',
	X = 1244.191  mm,	Y = 24.046  mm,	Z = -244.969  mm,
	W = 0.000 deg,	P = 30.000 deg,	R = -177.690 deg
};
P[259]{
   GP1:
	UF : 0, UT : 1,		CONFIG : 'N U T, 0, 0, 0',
	X = 1243.757  mm,	Y = 22.938  mm,	Z = -245.104  mm,
	W = 0.000 deg,	P = 30.000 deg,	R = -176.846 deg
};
P[260]{
   GP1:
	UF : 0, UT : 1,		CONFIG : 'N U T, 0, 0, 0',
	X = 1243.436  mm,	Y = 22.077  mm,	Z = -245.087  mm,
	W = 0.000 deg,	P = 30.000 deg,	R = -176.846 deg
};
P[261]{
   GP1:
	UF : 0, UT : 1,		CONFIG : 'N U T, 0, 0, 0',
	X = 1243.326  mm,	Y = 24.073  mm,	Z = -245.054  mm,
	W = 0.000 deg,	P = 30.000 deg,	R = -176.846 deg
};
P[262]{
   GP1:
	UF : 0, UT : 1,		CONFIG : 'N U T, 0, 0, 0',
	X = 1243.216  mm,	Y = 26.070  mm,	Z = -245.022  mm,
	W = 0.000 deg,	P = 30.000 deg,	R = -176.846 deg
};
P[263]{
   GP1:
	UF : 0, UT : 1,		CONFIG : 'N U T, 0, 0, 0',
	X = 1243.106  mm,	Y = 28.067  mm,	Z = -244.989  mm,
	W = 0.000 deg,	P = 30.000 deg,	R = -176.846 deg
};
P[264]{
   GP1:
	UF : 0, UT : 1,		CONFIG : 'N U T, 0, 0, 0',
	X = 1242.996  mm,	Y = 30.063  mm,	Z = -244.956  mm,
	W = 0.000 deg,	P = 30.000 deg,	R = -176.846 deg
};
P[265]{
   GP1:
	UF : 0, UT : 1,		CONFIG : 'N U T, 0, 0, 0',
	X = 1242.886  mm,	Y = 32.060  mm,	Z = -244.924  mm,
	W = 0.000 deg,	P = 30.000 deg,	R = -176.846 deg
};
P[266]{
   GP1:
	UF : 0, UT : 1,		CONFIG : 'N U T, 0, 0, 0',
	X = 1242.776  mm,	Y = 34.057  mm,	Z = -244.891  mm,
	W = 0.000 deg,	P = 30.000 deg,	R = -176.846 deg
};
P[267]{
   GP1:
	UF : 0, UT : 1,		CONFIG : 'N U T, 0, 0, 0',
	X = 1242.666  mm,	Y = 36.054  mm,	Z = -244.858  mm,
	W = 0.000 deg,	P = 30.000 deg,	R = -176.846 deg
};
P[268]{
   GP1:
	UF : 0, UT : 1,		CONFIG : 'N U T, 0, 0, 0',
	X = 1242.556  mm,	Y = 38.050  mm,	Z = -244.826  mm,
	W = 0.000 deg,	P = 30.000 deg,	R = -176.846 deg
};
P[269]{
   GP1:
	UF : 0, UT : 1,		CONFIG : 'N U T, 0, 0, 0',
	X = 1242.446  mm,	Y = 40.047  mm,	Z = -244.793  mm,
	W = 0.000 deg,	P = 30.000 deg,	R = -176.846 deg
};
P[270]{
   GP1:
	UF : 0, UT : 1,		CONFIG : 'N U T, 0, 0, 0',
	X = 1242.336  mm,	Y = 42.044  mm,	Z = -244.761  mm,
	W = 0.000 deg,	P = 30.000 deg,	R = -176.846 deg
};
P[271]{
   GP1:
	UF : 0, UT : 1,		CONFIG : 'N U T, 0, 0, 0',
	X = 1242.226  mm,	Y = 44.040  mm,	Z = -244.728  mm,
	W = 0.000 deg,	P = 30.000 deg,	R = -176.846 deg
};
P[272]{
   GP1:
	UF : 0, UT : 1,		CONFIG : 'N U T, 0, 0, 0',
	X = 1242.116  mm,	Y = 46.037  mm,	Z = -244.695  mm,
	W = 0.000 deg,	P = 30.000 deg,	R = -176.846 deg
};
P[273]{
   GP1:
	UF : 0, UT : 1,		CONFIG : 'N U T, 0, 0, 0',
	X = 1242.006  mm,	Y = 48.034  mm,	Z = -244.663  mm,
	W = 0.000 deg,	P = 30.000 deg,	R = -176.846 deg
};
P[274]{
   GP1:
	UF : 0, UT : 1,		CONFIG : 'N U T, 0, 0, 0',
	X = 1241.896  mm,	Y = 50.031  mm,	Z = -244.630  mm,
	W = 0.000 deg,	P = 30.000 deg,	R = -176.846 deg
};
P[275]{
   GP1:
	UF : 0, UT : 1,		CONFIG : 'N U T, 0, 0, 0',
	X = 1241.786  mm,	Y = 52.027  mm,	Z = -244.597  mm,
	W = 0.000 deg,	P = 30.000 deg,	R = -176.846 deg
};
P[276]{
   GP1:
	UF : 0, UT : 1,		CONFIG : 'N U T, 0, 0, 0',
	X = 1241.676  mm,	Y = 54.024  mm,	Z = -244.565  mm,
	W = 0.000 deg,	P = 30.000 deg,	R = -176.846 deg
};
P[277]{
   GP1:
	UF : 0, UT : 1,		CONFIG : 'N U T, 0, 0, 0',
	X = 1241.566  mm,	Y = 56.021  mm,	Z = -244.532  mm,
	W = 0.000 deg,	P = 30.000 deg,	R = -176.846 deg
};
P[278]{
   GP1:
	UF : 0, UT : 1,		CONFIG : 'N U T, 0, 0, 0',
	X = 1241.456  mm,	Y = 58.017  mm,	Z = -244.500  mm,
	W = 0.000 deg,	P = 30.000 deg,	R = -176.846 deg
};
P[279]{
   GP1:
	UF : 0, UT : 1,		CONFIG : 'N U T, 0, 0, 0',
	X = 1241.346  mm,	Y = 60.014  mm,	Z = -244.467  mm,
	W = 0.000 deg,	P = 30.000 deg,	R = -176.846 deg
};
P[280]{
   GP1:
	UF : 0, UT : 1,		CONFIG : 'N U T, 0, 0, 0',
	X = 1241.236  mm,	Y = 62.011  mm,	Z = -244.434  mm,
	W = 0.000 deg,	P = 30.000 deg,	R = -176.846 deg
};
P[281]{
   GP1:
	UF : 0, UT : 1,		CONFIG : 'N U T, 0, 0, 0',
	X = 1241.126  mm,	Y = 64.007  mm,	Z = -244.402  mm,
	W = 0.000 deg,	P = 30.000 deg,	R = -176.846 deg
};
P[282]{
   GP1:
	UF : 0, UT : 1,		CONFIG : 'N U T, 0, 0, 0',
	X = 1241.015  mm,	Y = 66.004  mm,	Z = -244.369  mm,
	W = 0.000 deg,	P = 30.000 deg,	R = -176.846 deg
};
P[283]{
   GP1:
	UF : 0, UT : 1,		CONFIG : 'N U T, 0, 0, 0',
	X = 1240.905  mm,	Y = 68.001  mm,	Z = -244.336  mm,
	W = 0.000 deg,	P = 30.000 deg,	R = -176.846 deg
};
P[284]{
   GP1:
	UF : 0, UT : 1,		CONFIG : 'N U T, 0, 0, 0',
	X = 1240.795  mm,	Y = 69.998  mm,	Z = -244.304  mm,
	W = 0.000 deg,	P = 30.000 deg,	R = -172.479 deg
};
P[285]{
   GP1:
	UF : 0, UT : 1,		CONFIG : 'N U T, 0, 0, 0',
	X = 1240.685  mm,	Y = 71.994  mm,	Z = -244.271  mm,
	W = 0.000 deg,	P = 30.000 deg,	R = -164.076 deg
};
P[286]{
   GP1:
	UF : 0, UT : 1,		CONFIG : 'N U T, 0, 0, 0',
	X = 1240.575  mm,	Y = 73.991  mm,	Z = -244.239  mm,
	W = 0.000 deg,	P = 30.000 deg,	R = -155.673 deg
};
P[287]{
   GP1:
	UF : 0, UT : 1,		CONFIG : 'N U T, 0, 0, 0',
	X = 1240.465  mm,	Y = 75.988  mm,	Z = -244.206  mm,
	W = 0.000 deg,	P = 30.000 deg,	R = -147.270 deg
};
P[288]{
   GP1:
	UF : 0, UT : 1,		CONFIG : 'N U T, 0, 0, 0',
	X = 1240.355  mm,	Y = 77.984  mm,	Z = -244.173  mm,
	W = 0.000 deg,	P = 30.000 deg,	R = -138.866 deg
};
P[289]{
   GP1:
	UF : 0, UT : 1,		CONFIG : 'N U T, 0, 0, 0',
	X = 1240.325  mm,	Y = 79.104  mm,	Z = -244.146  mm,
	W = 0.000 deg,	P = 30.000 deg,	R = -134.830 deg
};
P[290]{
   GP1:
	UF : 0, UT : 1,		CONFIG : 'N U T, 0, 0, 0',
	X = 1241.503  mm,	Y = 76.613  mm,	Z = -244.098  mm,
	W = 0.000 deg,	P = 30.000 deg,	R = -134.830 deg
};
P[291]{
   GP1:
	UF : 0, UT : 1,		CONFIG : 'N U T, 0, 0, 0',
	X = 1240.101  mm,	Y = 78.007  mm,	Z = -243.799  mm,
	W = 0.000 deg,	P = 30.000 deg,	R = -134.830 deg
};
P[292]{
   GP1:
	UF : 0, UT : 1,		CONFIG : 'N U T, 0, 0, 0',
	X = 1238.698  mm,	Y = 79.401  mm,	Z = -243.501  mm,
	W = 0.000 deg,	P = 30.000 deg,	R = -134.830 deg
};
P[293]{
   GP1:
	UF : 0, UT : 1,		CONFIG : 'N U T, 0, 0, 0',
	X = 1237.296  mm,	Y = 80.795  mm,	Z = -243.203  mm,
	W = 0.000 deg,	P = 30.000 deg,	R = -134.830 deg
};
P[294]{
   GP1:
	UF : 0, UT : 1,		CONFIG : 'N U T, 0, 0, 0',
	X = 1235.893  mm,	Y = 82.190  mm,	Z = -242.904  mm,
	W = 0.000 deg,	P = 30.000 deg,	R = -134.830 deg
};
P[295]{
   GP1:
	UF : 0, UT : 1,		CONFIG : 'N U T, 0, 0, 0',
	X = 1234.491  mm,	Y = 83.584  mm,	Z = -242.606  mm,
	W = 0.000 deg,	P = 30.000 deg,	R = -134.830 deg
};
P[296]{
   GP1:
	UF : 0, UT : 1,		CONFIG : 'N U T, 0, 0, 0',
	X = 1233.088  mm,	Y = 84.978  mm,	Z = -242.308  mm,
	W = 0.000 deg,	P = 30.000 deg,	R = -134.830 deg
};
P[297]{
   GP1:
	UF : 0, UT : 1,		CONFIG : 'N U T, 0, 0, 0',
	X = 1231.686  mm,	Y = 86.372  mm,	Z = -242.009  mm,
	W = 0.000 deg,	P = 30.000 deg,	R = -134.830 deg
};
P[298]{
   GP1:
	UF : 0, UT : 1,		CONFIG : 'N U T, 0, 0, 0',
	X = 1230.283  mm,	Y = 87.766  mm,	Z = -241.711  mm,
	W = 0.000 deg,	P = 30.000 deg,	R = -134.830 deg
};
P[299]{
   GP1:
	UF : 0, UT : 1,		CONFIG : 'N U T, 0, 0, 0',
	X = 1228.881  mm,	Y = 89.161  mm,	Z = -241.413  mm,
	W = 0.000 deg,	P = 30.000 deg,	R = -134.830 deg
};
P[300]{
   GP1:
	UF : 0, UT : 1,		CONFIG : 'N U T, 0, 0, 0',
	X = 1227.478  mm,	Y = 90.555  mm,	Z = -241.115  mm,
	W = 0.000 deg,	P = 30.000 deg,	R = -134.830 deg
};
P[301]{
   GP1:
	UF : 0, UT : 1,		CONFIG : 'N U T, 0, 0, 0',
	X = 1226.075  mm,	Y = 91.949  mm,	Z = -240.816  mm,
	W = 0.000 deg,	P = 30.000 deg,	R = -134.830 deg
};
P[302]{
   GP1:
	UF : 0, UT : 1,		CONFIG : 'N U T, 0, 0, 0',
	X = 1224.673  mm,	Y = 93.343  mm,	Z = -240.518  mm,
	W = 0.000 deg,	P = 30.000 deg,	R = -134.830 deg
};
P[303]{
   GP1:
	UF : 0, UT : 1,		CONFIG : 'N U T, 0, 0, 0',
	X = 1223.270  mm,	Y = 94.738  mm,	Z = -240.220  mm,
	W = 0.000 deg,	P = 30.000 deg,	R = -134.830 deg
};
P[304]{
   GP1:
	UF : 0, UT : 1,		CONFIG : 'N U T, 0, 0, 0',
	X = 1221.868  mm,	Y = 96.132  mm,	Z = -239.921  mm,
	W = 0.000 deg,	P = 30.000 deg,	R = -134.830 deg
};
P[305]{
   GP1:
	UF : 0, UT : 1,		CONFIG : 'N U T, 0, 0, 0',
	X = 1220.465  mm,	Y = 97.526  mm,	Z = -239.623  mm,
	W = 0.000 deg,	P = 30.000 deg,	R = -134.830 deg
};
P[306]{
   GP1:
	UF : 0, UT : 1,		CONFIG : 'N U T, 0, 0, 0',
	X = 1219.063  mm,	Y = 98.920  mm,	Z = -239.325  mm,
	W = 0.000 deg,	P = 30.000 deg,	R = -134.830 deg
};
P[307]{
   GP1:
	UF : 0, UT : 1,		CONFIG : 'N U T, 0, 0, 0',
	X = 1217.660  mm,	Y = 100.315  mm,	Z = -239.026  mm,
	W = 0.000 deg,	P = 30.000 deg,	R = -134.830 deg
};
P[308]{
   GP1:
	UF : 0, UT : 1,		CONFIG : 'N U T, 0, 0, 0',
	X = 1216.258  mm,	Y = 101.709  mm,	Z = -238.728  mm,
	W = 0.000 deg,	P = 30.000 deg,	R = -134.830 deg
};
P[309]{
   GP1:
	UF : 0, UT : 1,		CONFIG : 'N U T, 0, 0, 0',
	X = 1214.855  mm,	Y = 103.103  mm,	Z = -238.430  mm,
	W = 0.000 deg,	P = 30.000 deg,	R = -134.830 deg
};
P[310]{
   GP1:
	UF : 0, UT : 1,		CONFIG : 'N U T, 0, 0, 0',
	X = 1213.453  mm,	Y = 104.497  mm,	Z = -238.132  mm,
	W = 0.000 deg,	P = 30.000 deg,	R = -134.830 deg
};
P[311]{
   GP1:
	UF : 0, UT : 1,		CONFIG : 'N U T, 0, 0, 0',
	X = 1212.050  mm,	Y = 105.892  mm,	Z = -237.833  mm,
	W = 0.000 deg,	P = 30.000 deg,	R = -145.194 deg
};
P[312]{
   GP1:
	UF : 0, UT : 1,		CONFIG : 'N U T, 0, 0, 0',
	X = 1210.647  mm,	Y = 107.286  mm,	Z = -237.535  mm,
	W = 0.000 deg,	P = 30.000 deg,	R = -154.114 deg
};
P[313]{
   GP1:
	UF : 0, UT : 1,		CONFIG : 'N U T, 0, 0, 0',
	X = 1209.245  mm,	Y = 108.680  mm,	Z = -237.237  mm,
	W = 0.000 deg,	P = 30.000 deg,	R = -163.035 deg
};
P[314]{
   GP1:
	UF : 0, UT : 1,		CONFIG : 'N U T, 0, 0, 0',
	X = 1207.842  mm,	Y = 110.074  mm,	Z = -236.938  mm,
	W = 0.000 deg,	P = 30.000 deg,	R = -171.955 deg
};
P[315]{
   GP1:
	UF : 0, UT : 1,		CONFIG : 'N U T, 0, 0, 0',
	X = 1206.440  mm,	Y = 111.468  mm,	Z = -236.640  mm,
	W = 0.000 deg,	P = 30.000 deg,	R = -179.430 deg
};
P[316]{
   GP1:
	UF : 0, UT : 1,		CONFIG : 'N U T, 0, 0, 0',
	X = 1204.749  mm,	Y = 114.525  mm,	Z = -236.582  mm,
	W = 0.000 deg,	P = 30.000 deg,	R = -179.430 deg
};
P[317]{
   GP1:
	UF : 0, UT : 1,		CONFIG : 'N U T, 0, 0, 0',
	X = 1204.675  mm,	Y = 116.846  mm,	Z = -236.566  mm,
	W = 0.000 deg,	P = 30.000 deg,	R = -179.430 deg
};
P[318]{
   GP1:
	UF : 0, UT : 1,		CONFIG : 'N U T, 0, 0, 0',
	X = 1204.655  mm,	Y = 118.846  mm,	Z = -236.547  mm,
	W = 0.000 deg,	P = 30.000 deg,	R = -179.430 deg
};
P[319]{
   GP1:
	UF : 0, UT : 1,		CONFIG : 'N U T, 0, 0, 0',
	X = 1204.635  mm,	Y = 120.846  mm,	Z = -236.528  mm,
	W = 0.000 deg,	P = 30.000 deg,	R = -179.430 deg
};
P[320]{
   GP1:
	UF : 0, UT : 1,		CONFIG : 'N U T, 0, 0, 0',
	X = 1204.615  mm,	Y = 122.846  mm,	Z = -236.509  mm,
	W = 0.000 deg,	P = 30.000 deg,	R = -179.430 deg
};
P[321]{
   GP1:
	UF : 0, UT : 1,		CONFIG : 'N U T, 0, 0, 0',
	X = 1204.595  mm,	Y = 124.845  mm,	Z = -236.490  mm,
	W = 0.000 deg,	P = 30.000 deg,	R = -179.430 deg
};
P[322]{
   GP1:
	UF : 0, UT : 1,		CONFIG : 'N U T, 0, 0, 0',
	X = 1204.576  mm,	Y = 126.845  mm,	Z = -236.471  mm,
	W = 0.000 deg,	P = 30.000 deg,	R = -179.430 deg
};
P[323]{
   GP1:
	UF : 0, UT : 1,		CONFIG : 'N U T, 0, 0, 0',
	X = 1204.556  mm,	Y = 128.845  mm,	Z = -236.452  mm,
	W = 0.000 deg,	P = 30.000 deg,	R = -179.430 deg
};
P[324]{
   GP1:
	UF : 0, UT : 1,		CONFIG : 'N U T, 0, 0, 0',
	X = 1204.536  mm,	Y = 130.845  mm,	Z = -236.433  mm,
	W = 0.000 deg,	P = 30.000 deg,	R = -179.430 deg
};
P[325]{
   GP1:
	UF : 0, UT : 1,		CONFIG : 'N U T, 0, 0, 0',
	X = 1204.516  mm,	Y = 132.845  mm,	Z = -236.414  mm,
	W = 0.000 deg,	P = 30.000 deg,	R = -179.430 deg
};
P[326]{
   GP1:
	UF : 0, UT : 1,		CONFIG : 'N U T, 0, 0, 0',
	X = 1204.496  mm,	Y = 134.844  mm,	Z = -236.395  mm,
	W = 0.000 deg,	P = 30.000 deg,	R = -179.430 deg
};
P[327]{
   GP1:
	UF : 0, UT : 1,		CONFIG : 'N U T, 0, 0, 0',
	X = 1204.476  mm,	Y = 136.844  mm,	Z = -236.376  mm,
	W = 0.000 deg,	P = 30.000 deg,	R = -179.430 deg
};
P[328]{
   GP1:
	UF : 0, UT : 1,		CONFIG : 'N U T, 0, 0, 0',
	X = 1204.456  mm,	Y = 138.844  mm,	Z = -236.356  mm,
	W = 0.000 deg,	P = 30.000 deg,	R = -179.430 deg
};
P[329]{
   GP1:
	UF : 0, UT : 1,		CONFIG : 'N U T, 0, 0, 0',
	X = 1204.436  mm,	Y = 140.844  mm,	Z = -236.337  mm,
	W = 0.000 deg,	P = 30.000 deg,	R = -179.430 deg
};
P[330]{
   GP1:
	UF : 0, UT : 1,		CONFIG : 'N U T, 0, 0, 0',
	X = 1204.416  mm,	Y = 142.844  mm,	Z = -236.318  mm,
	W = 0.000 deg,	P = 30.000 deg,	R = -179.430 deg
};
P[331]{
   GP1:
	UF : 0, UT : 1,		CONFIG : 'N U T, 0, 0, 0',
	X = 1204.397  mm,	Y = 144.844  mm,	Z = -236.299  mm,
	W = 0.000 deg,	P = 30.000 deg,	R = -179.430 deg
};
P[332]{
   GP1:
	UF : 0, UT : 1,		CONFIG : 'N U T, 0, 0, 0',
	X = 1204.377  mm,	Y = 146.843  mm,	Z = -236.280  mm,
	W = 0.000 deg,	P = 30.000 deg,	R = -179.430 deg
};
P[333]{
   GP1:
	UF : 0, UT : 1,		CONFIG : 'N U T, 0, 0, 0',
	X = 1204.357  mm,	Y = 148.843  mm,	Z = -236.261  mm,
	W = 0.000 deg,	P = 30.000 deg,	R = -179.430 deg
};
P[334]{
   GP1:
	UF : 0, UT : 1,		CONFIG : 'N U T, 0, 0, 0',
	X = 1204.337  mm,	Y = 150.843  mm,	Z = -236.242  mm,
	W = 0.000 deg,	P = 30.000 deg,	R = -179.430 deg
};
P[335]{
   GP1:
	UF : 0, UT : 1,		CONFIG : 'N U T, 0, 0, 0',
	X = 1204.317  mm,	Y = 152.843  mm,	Z = -236.223  mm,
	W = 0.000 deg,	P = 30.000 deg,	R = -179.430 deg
};
P[336]{
   GP1:
	UF : 0, UT : 1,		CONFIG : 'N U T, 0, 0, 0',
	X = 1204.297  mm,	Y = 154.843  mm,	Z = -236.204  mm,
	W = 0.000 deg,	P = 30.000 deg,	R = -179.430 deg
};
P[337]{
   GP1:
	UF : 0, UT : 1,		CONFIG : 'N U T, 0, 0, 0',
	X = 1204.277  mm,	Y = 156.842  mm,	Z = -236.185  mm,
	W = 0.000 deg,	P = 30.000 deg,	R = -179.430 deg
};
P[338]{
   GP1:
	UF : 0, UT : 1,		CONFIG : 'N U T, 0, 0, 0',
	X = 1204.257  mm,	Y = 158.842  mm,	Z = -236.166  mm,
	W = 0.000 deg,	P = 30.000 deg,	R = -179.430 deg
};
P[339]{
   GP1:
	UF : 0, UT : 1,		CONFIG : 'N U T, 0, 0, 0',
	X = 1204.237  mm,	Y = 160.842  mm,	Z = -236.147  mm,
	W = 0.000 deg,	P = 30.000 deg,	R = -179.430 deg
};
P[340]{
   GP1:
	UF : 0, UT : 1,		CONFIG : 'N U T, 0, 0, 0',
	X = 1204.218  mm,	Y = 162.842  mm,	Z = -236.128  mm,
	W = 0.000 deg,	P = 30.000 deg,	R = -179.430 deg
};
P[341]{
   GP1:
	UF : 0, UT : 1,		CONFIG : 'N U T, 0, 0, 0',
	X = 1204.198  mm,	Y = 164.842  mm,	Z = -236.108  mm,
	W = 0.000 deg,	P = 30.000 deg,	R = 173.412 deg
};
P[342]{
   GP1:
	UF : 0, UT : 1,		CONFIG : 'N U T, 0, 0, 0',
	X = 1204.178  mm,	Y = 166.841  mm,	Z = -236.089  mm,
	W = 0.000 deg,	P = 30.000 deg,	R = 164.516 deg
};
P[343]{
   GP1:
	UF : 0, UT : 1,		CONFIG : 'N U T, 0, 0, 0',
	X = 1204.158  mm,	Y = 168.841  mm,	Z = -236.070  mm,
	W = 0.000 deg,	P = 30.000 deg,	R = 155.620 deg
};
P[344]{
   GP1:
	UF : 0, UT : 1,		CONFIG : 'N U T, 0, 0, 0',
	X = 1204.138  mm,	Y = 170.841  mm,	Z = -236.051  mm,
	W = 0.000 deg,	P = 30.000 deg,	R = 146.724 deg
};
P[345]{
   GP1:
	UF : 0, UT : 1,		CONFIG : 'N U T, 0, 0, 0',
	X = 1204.118  mm,	Y = 172.841  mm,	Z = -236.032  mm,
	W = 0.000 deg,	P = 30.000 deg,	R = 137.828 deg
};
P[346]{
   GP1:
	UF : 0, UT : 1,		CONFIG : 'N U T, 0, 0, 0',
	X = 1204.125  mm,	Y = 175.080  mm,	Z = -236.016  mm,
	W = 0.000 deg,	P = 30.000 deg,	R = 136.089 deg
};
P[347]{
   GP1:
	UF : 0, UT : 1,		CONFIG : 'N U T, 0, 0, 0',
	X = 1205.703  mm,	Y = 178.272  mm,	Z = -236.060  mm,
	W = 0.000 deg,	P = 30.000 deg,	R = 136.089 deg
};
P[348]{
   GP1:
	UF : 0, UT : 1,		CONFIG : 'N U T, 0, 0, 0',
	X = 1207.075  mm,	Y = 179.697  mm,	Z = -236.357  mm,
	W = 0.000 deg,	P = 30.000 deg,	R = 136.089 deg
};
P[349]{
   GP1:
	UF : 0, UT : 1,		CONFIG : 'N U T, 0, 0, 0',
	X = 1208.447  mm,	Y = 181.122  mm,	Z = -236.654  mm,
	W = 0.000 deg,	P = 30.000 deg,	R = 136.089 deg
};
P[350]{
   GP1:
	UF : 0, UT : 1,		CONFIG : 'N U T, 0, 0, 0',
	X = 1209.818  mm,	Y = 182.547  mm,	Z = -236.951  mm,
	W = 0.000 deg,	P = 30.000 deg,	R = 136.089 deg
};
P[351]{
   GP1:
	UF : 0, UT : 1,		CONFIG : 'N U T, 0, 0, 0',
	X = 1211.190  mm,	Y = 183.972  mm,	Z = -237.248  mm,
	W = 0.000 deg,	P = 30.000 deg,	R = 136.089 deg
};
P[352]{
   GP1:
	UF : 0, UT : 1,		CONFIG : 'N U T, 0, 0, 0',
	X = 1212.562  mm,	Y = 185.397  mm,	Z = -237.544  mm,
	W = 0.000 deg,	P = 30.000 deg,	R = 136.089 deg
};
P[353]{
   GP1:
	UF : 0, UT : 1,		CONFIG : 'N U T, 0, 0, 0',
	X = 1213.934  mm,	Y = 186.822  mm,	Z = -237.841  mm,
	W = 0.000 deg,	P = 30.000 deg,	R = 136.089 deg
};
P[354]{
   GP1:
	UF : 0, UT : 1,		CONFIG : 'N U T, 0, 0, 0',
	X = 1215.305  mm,	Y = 188.247  mm,	Z = -238.138  mm,
	W = 0.000 deg,	P = 30.000 deg,	R = 136.089 deg
};
P[355]{
   GP1:
	UF : 0, UT : 1,		CONFIG : 'N U T, 0, 0, 0',
	X = 1216.677  mm,	Y = 189.671  mm,	Z = -238.435  mm,
	W = 0.000 deg,	P = 30.000 deg,	R = 136.089 deg
};
P[356]{
   GP1:
	UF : 0, UT : 1,		CONFIG : 'N U T, 0, 0, 0',
	X = 1218.049  mm,	Y = 191.096  mm,	Z = -238.732  mm,
	W = 0.000 deg,	P = 30.000 deg,	R = 136.089 deg
};
P[357]{
   GP1:
	UF : 0, UT : 1,		CONFIG : 'N U T, 0, 0, 0',
	X = 1219.421  mm,	Y = 192.521  mm,	Z = -239.029  mm,
	W = 0.000 deg,	P = 30.000 deg,	R = 136.089 deg
};
P[358]{
   GP1:
	UF : 0, UT : 1,		CONFIG : 'N U T, 0, 0, 0',
	X = 1220.792  mm,	Y = 193.946  mm,	Z = -239.325  mm,
	W = 0.000 deg,	P = 30.000 deg,	R = 136.089 deg
};
P[359]{
   GP1:
	UF : 0, UT : 1,		CONFIG : 'N U T, 0, 0, 0',
	X = 1222.164  mm,	Y = 195.371  mm,	Z = -239.622  mm,
	W = 0.000 deg,	P = 30.000 deg,	R = 136.089 deg
};
P[360]{
   GP1:
	UF : 0, UT : 1,		CONFIG : 'N U T, 0, 0, 0',
	X = 1223.536  mm,	Y = 196.796  mm,	Z = -239.919  mm,
	W = 0.000 deg,	P = 30.000 deg,	R = 136.089 deg
};
P[361]{
   GP1:
	UF : 0, UT : 1,		CONFIG : 'N U T, 0, 0, 0',
	X = 1224.907  mm,	Y = 198.221  mm,	Z = -240.216  mm,
	W = 0.000 deg,	P = 30.000 deg,	R = 136.089 deg
};
P[362]{
   GP1:
	UF : 0, UT : 1,		CONFIG : 'N U T, 0, 0, 0',
	X = 1226.279  mm,	Y = 199.646  mm,	Z = -240.513  mm,
	W = 0.000 deg,	P = 30.000 deg,	R = 136.089 deg
};
P[363]{
   GP1:
	UF : 0, UT : 1,		CONFIG : 'N U T, 0, 0, 0',
	X = 1227.651  mm,	Y = 201.070  mm,	Z = -240.810  mm,
	W = 0.000 deg,	P = 30.000 deg,	R = 136.089 deg
};
P[364]{
   GP1:
	UF : 0, UT : 1,		CONFIG : 'N U T, 0, 0, 0',
	X = 1229.023  mm,	Y = 202.495  mm,	Z = -241.106  mm,
	W = 0.000 deg,	P = 30.000 deg,	R = 136.089 deg
};
P[365]{
   GP1:
	UF : 0, UT : 1,		CONFIG : 'N U T, 0, 0, 0',
	X = 1230.394  mm,	Y = 203.920  mm,	Z = -241.403  mm,
	W = 0.000 deg,	P = 30.000 deg,	R = 136.089 deg
};
P[366]{
   GP1:
	UF : 0, UT : 1,		CONFIG : 'N U T, 0, 0, 0',
	X = 1231.766  mm,	Y = 205.345  mm,	Z = -241.700  mm,
	W = 0.000 deg,	P = 30.000 deg,	R = 137.398 deg
};
P[367]{
   GP1:
	UF : 0, UT : 1,		CONFIG : 'N U T, 0, 0, 0',
	X = 1233.138  mm,	Y = 206.770  mm,	Z = -241.997  mm,
	W = 0.000 deg,	P = 30.000 deg,	R = 146.189 deg
};
P[368]{
   GP1:
	UF : 0, UT : 1,		CONFIG : 'N U T, 0, 0, 0',
	X = 1234.510  mm,	Y = 208.195  mm,	Z = -242.294  mm,
	W = 0.000 deg,	P = 30.000 deg,	R = 154.980 deg
};
P[369]{
   GP1:
	UF : 0, UT : 1,		CONFIG : 'N U T, 0, 0, 0',
	X = 1235.881  mm,	Y = 209.620  mm,	Z = -242.591  mm,
	W = 0.000 deg,	P = 30.000 deg,	R = 163.771 deg
};
P[370]{
   GP1:
	UF : 0, UT : 1,		CONFIG : 'N U T, 0, 0, 0',
	X = 1237.253  mm,	Y = 211.044  mm,	Z = -242.887  mm,
	W = 0.000 deg,	P = 30.000 deg,	R = 172.562 deg
};
P[371]{
   GP1:
	UF : 0, UT : 1,		CONFIG : 'N U T, 0, 0, 0',
	X = 1238.625  mm,	Y = 212.469  mm,	Z = -243.184  mm,
	W = 0.000 deg,	P = 30.000 deg,	R = -179.957 deg
};
P[372]{
   GP1:
	UF : 0, UT : 1,		CONFIG : 'N U T, 0, 0, 0',
	X = 1238.519  mm,	Y = 211.996  mm,	Z = -243.357  mm,
	W = 0.000 deg,	P = 30.000 deg,	R = -179.957 deg
};
P[373]{
   GP1:
	UF : 0, UT : 1,		CONFIG : 'N U T, 0, 0, 0',
	X = 1238.026  mm,	Y = 210.663  mm,	Z = -243.359  mm,
	W = 0.000 deg,	P = 30.000 deg,	R = -179.957 deg
};
P[374]{
   GP1:
	UF : 0, UT : 1,		CONFIG : 'N U T, 0, 0, 0',
	X = 1238.024  mm,	Y = 212.663  mm,	Z = -243.362  mm,
	W = 0.000 deg,	P = 30.000 deg,	R = -179.957 deg
};
P[375]{
   GP1:
	UF : 0, UT : 1,		CONFIG : 'N U T, 0, 0, 0',
	X = 1238.023  mm,	Y = 214.663  mm,	Z = -243.365  mm,
	W = 0.000 deg,	P = 30.000 deg,	R = -179.957 deg
};
P[376]{
   GP1:
	UF : 0, UT : 1,		CONFIG : 'N U T, 0, 0, 0',
	X = 1238.021  mm,	Y = 216.663  mm,	Z = -243.368  mm,
	W = 0.000 deg,	P = 30.000 deg,	R = -179.957 deg
};
P[377]{
   GP1:
	UF : 0, UT : 1,		CONFIG : 'N U T, 0, 0, 0',
	X = 1238.020  mm,	Y = 218.663  mm,	Z = -243.371  mm,
	W = 0.000 deg,	P = 30.000 deg,	R = -179.957 deg
};
P[378]{
   GP1:
	UF : 0, UT : 1,		CONFIG : 'N U T, 0, 0, 0',
	X = 1238.018  mm,	Y = 220.663  mm,	Z = -243.374  mm,
	W = 0.000 deg,	P = 30.000 deg,	R = -179.957 deg
};
P[379]{
   GP1:
	UF : 0, UT : 1,		CONFIG : 'N U T, 0, 0, 0',
	X = 1238.017  mm,	Y = 221.828  mm,	Z = -243.376  mm,
	W = 0.000 deg,	P = 30.000 deg,	R = -179.957 deg
};
/END
